C05358=1022.023,281.198,-131.885,170.057,49.076,159.456
C05359=1022.016,280.949,-131.855,170.053,49.079,159.456
C05360=1022.009,280.702,-131.824,170.047,49.082,159.456
C05361=1022.003,280.454,-131.794,170.043,49.086,159.456
C05362=1021.996,280.205,-131.763,170.039,49.089,159.456
C05363=1021.991,279.958,-131.733,170.034,49.092,159.456
C05364=1021.984,279.710,-131.701,170.030,49.095,159.456
C05365=1021.977,279.462,-131.671,170.024,49.099,159.456
C05366=1021.971,279.214,-131.641,170.020,49.102,159.456
C05367=1021.965,278.966,-131.610,170.015,49.105,159.456
C05368=1021.959,278.749,-131.583,170.011,49.108,159.456
C05369=1021.953,278.533,-131.557,170.008,49.111,159.456
C05370=1021.948,278.315,-131.529,170.003,49.114,159.456
C05371=1021.942,278.099,-131.503,169.999,49.117,159.456
C05372=1021.937,277.882,-131.477,169.995,49.120,159.456
C05373=1021.931,277.665,-131.450,169.991,49.122,159.456
C05374=1021.926,277.449,-131.423,169.987,49.126,159.457
C05375=1021.921,277.232,-131.396,169.983,49.129,159.457
C05376=1021.914,276.984,-131.366,169.979,49.132,159.457
C05377=1021.908,276.736,-131.336,169.974,49.136,159.457
C05378=1021.901,276.488,-131.306,169.969,49.138,159.457
C05379=1021.895,276.240,-131.275,169.964,49.142,159.457
C05380=1021.888,275.992,-131.244,169.960,49.146,159.457
C05381=1021.882,275.744,-131.215,169.955,49.149,159.457
C05382=1021.876,275.495,-131.185,169.951,49.153,159.457
C05383=1021.869,275.247,-131.155,169.946,49.156,159.457
C05384=1021.863,275.000,-131.125,169.942,49.160,159.457
C05385=1021.856,274.751,-131.094,169.938,49.163,159.457
C05386=1021.850,274.504,-131.064,169.933,49.167,159.457
C05387=1021.843,274.255,-131.034,169.929,49.170,159.457
C05388=1021.837,274.008,-131.004,169.923,49.173,159.457
C05389=1021.831,273.759,-130.974,169.919,49.177,159.458
C05390=1021.825,273.511,-130.944,169.914,49.181,159.458
C05391=1021.818,273.263,-130.914,169.910,49.184,159.458
C05392=1021.812,273.015,-130.883,169.905,49.187,159.458
C05393=1021.806,272.767,-130.853,169.901,49.191,159.458
C05394=1021.799,272.518,-130.824,169.896,49.195,159.458
C05395=1021.793,272.271,-130.794,169.892,49.198,159.458
C05396=1021.786,272.022,-130.763,169.887,49.202,159.458
C05397=1021.780,271.774,-130.734,169.883,49.206,159.458
C05398=1021.774,271.526,-130.704,169.879,49.209,159.459
C05399=1021.767,271.278,-130.674,169.874,49.213,159.459
C05400=1021.761,271.030,-130.644,169.870,49.216,159.459
C05401=1021.755,270.782,-130.614,169.865,49.220,159.459
C05402=1021.748,270.533,-130.584,169.861,49.223,159.459
C05403=1021.742,270.285,-130.555,169.856,49.227,159.459
C05404=1021.736,270.038,-130.525,169.852,49.231,159.459
C05405=1021.729,269.789,-130.495,169.847,49.235,159.459
C05406=1021.723,269.541,-130.465,169.843,49.238,159.460
C05407=1021.717,269.293,-130.435,169.838,49.242,159.460
C05408=1021.710,269.045,-130.405,169.834,49.246,159.460
C05409=1021.704,268.796,-130.376,169.829,49.250,159.460
C05410=1021.697,268.549,-130.346,169.825,49.253,159.460
C05411=1021.692,268.300,-130.317,169.821,49.257,159.460
C05412=1021.685,268.052,-130.287,169.816,49.260,159.460
C05413=1021.679,267.804,-130.258,169.812,49.264,159.460
C05414=1021.673,267.556,-130.227,169.807,49.268,159.461
C05415=1021.666,267.307,-130.198,169.803,49.271,159.461
C05416=1021.660,267.059,-130.169,169.799,49.276,159.461
C05417=1021.653,266.812,-130.139,169.795,49.279,159.461
C05418=1021.648,266.563,-130.109,169.790,49.283,159.461
C05419=1021.641,266.315,-130.080,169.786,49.287,159.461
C05420=1021.634,266.067,-130.050,169.781,49.291,159.462
C05421=1021.628,265.819,-130.021,169.777,49.294,159.462
C05422=1021.622,265.570,-129.992,169.772,49.298,159.462
C05423=1021.616,265.323,-129.962,169.768,49.302,159.462
C05424=1021.609,265.074,-129.932,169.763,49.306,159.462
C05425=1021.603,264.826,-129.903,169.759,49.310,159.462
C05426=1021.596,264.578,-129.874,169.754,49.314,159.463
C05427=1021.590,264.330,-129.845,169.751,49.318,159.463
C05428=1021.585,264.116,-129.819,169.747,49.321,159.463
C05429=1021.579,263.901,-129.794,169.742,49.324,159.463
C05430=1021.573,263.686,-129.769,169.739,49.328,159.463
C05431=1021.568,263.472,-129.744,169.735,49.331,159.463
C05432=1021.563,263.258,-129.718,169.731,49.335,159.464
C05433=1021.557,263.044,-129.693,169.728,49.338,159.464
C05434=1021.552,262.829,-129.668,169.724,49.341,159.464
C05435=1021.547,262.615,-129.643,169.720,49.345,159.464
C05436=1021.541,262.366,-129.614,169.716,49.349,159.464
C05437=1021.534,262.118,-129.584,169.712,49.352,159.464
C05438=1021.528,261.869,-129.555,169.708,49.357,159.465
C05439=1021.521,261.621,-129.526,169.703,49.360,159.465
C05440=1021.515,261.373,-129.497,169.699,49.365,159.465
C05441=1021.508,261.126,-129.467,169.694,49.369,159.465
C05442=1021.503,260.877,-129.438,169.690,49.372,159.466
C05443=1021.497,260.629,-129.409,169.686,49.377,159.466
C05444=1021.490,260.381,-129.380,169.682,49.380,159.466
C05445=1021.485,260.132,-129.351,169.677,49.385,159.466
C05446=1021.478,259.884,-129.323,169.673,49.388,159.466
C05447=1021.471,259.636,-129.294,169.669,49.393,159.467
C05448=1021.464,259.387,-129.265,169.665,49.397,159.467
C05449=1021.457,259.140,-129.236,169.660,49.401,159.467
C05450=1021.452,258.891,-129.208,169.656,49.405,159.468
C05451=1021.445,258.643,-129.179,169.652,49.410,159.468
C05452=1021.438,258.395,-129.150,169.647,49.414,159.468
C05453=1021.432,258.147,-129.121,169.643,49.418,159.468
C05454=1021.426,257.898,-129.093,169.639,49.422,159.469
C05455=1021.420,257.650,-129.064,169.635,49.426,159.469
C05456=1021.413,257.402,-129.035,169.630,49.430,159.469
C05457=1021.407,257.153,-129.007,169.626,49.435,159.469
C05458=1021.401,256.905,-128.978,169.622,49.439,159.470
C05459=1021.394,256.657,-128.950,169.618,49.443,159.470
C05460=1021.388,256.409,-128.921,169.613,49.447,159.470
C05461=1021.381,256.160,-128.892,169.610,49.452,159.470
C05462=1021.375,255.912,-128.865,169.605,49.456,159.471
C05463=1021.369,255.664,-128.835,169.601,49.460,159.471
C05464=1021.362,255.416,-128.806,169.596,49.464,159.471
C05465=1021.356,255.167,-128.779,169.592,49.469,159.471
C05466=1021.349,254.919,-128.750,169.588,49.473,159.472
C05467=1021.343,254.670,-128.721,169.583,49.477,159.472
C05468=1021.337,254.422,-128.692,169.580,49.481,159.472
C05469=1021.330,254.174,-128.665,169.575,49.486,159.473
C05470=1021.324,253.926,-128.636,169.571,49.490,159.473
C05471=1021.318,253.677,-128.607,169.567,49.494,159.473
C05472=1021.311,253.429,-128.579,169.563,49.499,159.474
C05473=1021.305,253.180,-128.550,169.559,49.503,159.474
C05474=1021.299,252.932,-128.521,169.555,49.507,159.474
C05475=1021.292,252.684,-128.494,169.550,49.511,159.474
C05476=1021.286,252.436,-128.465,169.546,49.516,159.475
C05477=1021.280,252.187,-128.436,169.542,49.520,159.475
C05478=1021.273,251.939,-128.408,169.538,49.524,159.475
C05479=1021.267,251.690,-128.380,169.534,49.529,159.476
C05480=1021.262,251.442,-128.352,169.530,49.533,159.476
C05481=1021.255,251.195,-128.323,169.525,49.538,159.476
C05482=1021.249,250.946,-128.295,169.522,49.542,159.477
C05483=1021.243,250.698,-128.266,169.517,49.547,159.477
C05484=1021.236,250.449,-128.238,169.513,49.551,159.477
C05485=1021.230,250.200,-128.210,169.509,49.555,159.477
C05486=1021.224,249.952,-128.181,169.504,49.560,159.478
C05487=1021.218,249.705,-128.153,169.501,49.564,159.478
C05488=1021.212,249.489,-128.128,169.497,49.568,159.478
C05489=1021.208,249.274,-128.104,169.493,49.572,159.479
C05490=1021.202,249.058,-128.080,169.490,49.575,159.479
C05491=1021.197,248.843,-128.055,169.487,49.579,159.479
C05492=1021.191,248.629,-128.030,169.483,49.583,159.479
C05493=1021.186,248.413,-128.006,169.479,49.587,159.480
C05494=1021.180,248.198,-127.982,169.475,49.591,159.480
C05495=1021.175,247.983,-127.957,169.473,49.595,159.480
C05496=1021.169,247.734,-127.929,169.468,49.599,159.481
C05497=1021.163,247.485,-127.901,169.464,49.604,159.481
C05498=1021.156,247.237,-127.872,169.460,49.608,159.481
C05499=1021.151,246.989,-127.844,169.456,49.612,159.482
C05500=1021.144,246.741,-127.816,169.452,49.617,159.482
C05501=1021.138,246.492,-127.788,169.448,49.621,159.482
C05502=1021.133,246.243,-127.760,169.443,49.626,159.483
C05503=1021.126,245.996,-127.732,169.440,49.630,159.483
C05504=1021.120,245.747,-127.703,169.435,49.635,159.483
C05505=1021.114,245.499,-127.675,169.432,49.640,159.484
C05506=1021.108,245.251,-127.648,169.427,49.644,159.484
C05507=1021.102,245.002,-127.619,169.424,49.648,159.484
C05508=1021.096,244.753,-127.591,169.419,49.653,159.485
C05509=1021.090,244.506,-127.564,169.415,49.657,159.485
C05510=1021.084,244.257,-127.535,169.411,49.662,159.485
C05511=1021.078,244.008,-127.507,169.408,49.667,159.486
C05512=1021.072,243.761,-127.479,169.403,49.671,159.486
C05513=1021.066,243.512,-127.451,169.399,49.676,159.486
C05514=1021.060,243.263,-127.423,169.395,49.681,159.487
C05515=1021.054,243.015,-127.395,169.392,49.685,159.487
C05516=1021.048,242.767,-127.368,169.387,49.690,159.487
C05517=1021.041,242.518,-127.340,169.383,49.695,159.488
C05518=1021.036,242.270,-127.312,169.379,49.699,159.488
C05519=1021.029,242.022,-127.284,169.375,49.704,159.489
C05520=1021.023,241.773,-127.256,169.371,49.709,159.489
C05521=1021.017,241.525,-127.229,169.367,49.713,159.489
C05522=1021.010,241.277,-127.201,169.364,49.718,159.490
C05523=1021.005,241.028,-127.173,169.359,49.723,159.490
C05524=1020.998,240.780,-127.146,169.355,49.728,159.491
C05525=1020.992,240.531,-127.118,169.351,49.732,159.491
C05526=1020.986,240.283,-127.090,169.347,49.737,159.491
C05527=1020.980,240.035,-127.063,169.343,49.742,159.492
C05528=1020.973,239.786,-127.036,169.339,49.746,159.492
C05529=1020.968,239.538,-127.008,169.336,49.751,159.493
C05530=1020.961,239.289,-126.980,169.331,49.756,159.493
C05531=1020.955,239.042,-126.952,169.327,49.761,159.493
C05532=1020.949,238.793,-126.925,169.324,49.766,159.494
C05533=1020.942,238.544,-126.898,169.319,49.771,159.494
C05534=1020.937,238.295,-126.870,169.316,49.776,159.495
C05535=1020.931,238.047,-126.843,169.311,49.780,159.495
C05536=1020.924,237.799,-126.815,169.307,49.785,159.496
C05537=1020.918,237.550,-126.788,169.304,49.790,159.496
C05538=1020.911,237.302,-126.761,169.299,49.795,159.496
C05539=1020.906,237.053,-126.734,169.296,49.800,159.497
C05540=1020.899,236.805,-126.706,169.292,49.805,159.497
C05541=1020.893,236.557,-126.680,169.287,49.810,159.498
C05542=1020.886,236.308,-126.652,169.284,49.815,159.498
C05543=1020.881,236.059,-126.625,169.280,49.820,159.499
C05544=1020.875,235.811,-126.597,169.275,49.825,159.499
C05545=1020.869,235.563,-126.570,169.272,49.830,159.499
C05546=1020.862,235.314,-126.543,169.268,49.835,159.500
C05547=1020.857,235.066,-126.516,169.264,49.840,159.500
C05548=1020.851,234.847,-126.492,169.261,49.844,159.501
C05549=1020.845,234.629,-126.468,169.257,49.848,159.501
C05550=1020.840,234.410,-126.444,169.254,49.853,159.502
C05551=1020.834,234.192,-126.421,169.251,49.858,159.502
C05552=1020.828,233.974,-126.396,169.247,49.862,159.502
C05553=1020.823,233.756,-126.373,169.243,49.866,159.503
C05554=1020.818,233.537,-126.348,169.240,49.871,159.503
C05555=1020.813,233.319,-126.325,169.237,49.875,159.504
C05556=1020.807,233.070,-126.298,169.232,49.881,159.504
C05557=1020.800,232.822,-126.270,169.229,49.885,159.504
C05558=1020.794,232.574,-126.244,169.225,49.890,159.505
C05559=1020.788,232.324,-126.217,169.220,49.895,159.505
C05560=1020.782,232.077,-126.189,169.217,49.900,159.506
C05561=1020.776,231.828,-126.162,169.213,49.906,159.506
C05562=1020.770,231.579,-126.136,169.209,49.911,159.507
C05563=1020.763,231.330,-126.109,169.206,49.916,159.507
C05564=1020.757,231.083,-126.081,169.201,49.921,159.508
C05565=1020.752,230.834,-126.055,169.198,49.926,159.508
C05566=1020.745,230.585,-126.027,169.194,49.931,159.509
C05567=1020.739,230.337,-126.000,169.189,49.936,159.509
C05568=1020.733,230.088,-125.973,169.186,49.941,159.510
C05569=1020.727,229.840,-125.946,169.182,49.946,159.510
C05570=1020.721,229.592,-125.920,169.178,49.952,159.511
C05571=1020.715,229.342,-125.893,169.175,49.957,159.511
C05572=1020.708,229.095,-125.866,169.171,49.962,159.512
C05573=1020.702,228.847,-125.839,169.167,49.968,159.512
C05574=1020.696,228.598,-125.812,169.163,49.973,159.513
C05575=1020.690,228.349,-125.786,169.159,49.978,159.513
C05576=1020.684,228.101,-125.759,169.155,49.983,159.514
C05577=1020.678,227.852,-125.732,169.152,49.988,159.514
C05578=1020.672,227.604,-125.705,169.148,49.994,159.515
C05579=1020.666,227.354,-125.678,169.143,49.999,159.515
C05580=1020.659,227.106,-125.652,169.140,50.004,159.516
C05581=1020.653,226.858,-125.626,169.136,50.009,159.516
C05582=1020.648,226.610,-125.599,169.132,50.015,159.517
C05583=1020.641,226.361,-125.572,169.129,50.020,159.517
C05584=1020.635,226.113,-125.546,169.125,50.025,159.518
C05585=1020.629,225.864,-125.519,169.120,50.031,159.518
C05586=1020.622,225.615,-125.493,169.117,50.037,159.519
C05587=1020.616,225.367,-125.466,169.113,50.042,159.520
C05588=1020.610,225.119,-125.440,169.109,50.047,159.520
C05589=1020.603,224.870,-125.413,169.105,50.053,159.521
C05590=1020.598,224.622,-125.387,169.101,50.058,159.521
C05591=1020.592,224.373,-125.361,169.098,50.063,159.522
C05592=1020.585,224.124,-125.334,169.094,50.068,159.522
C05593=1020.579,223.876,-125.308,169.090,50.074,159.523
C05594=1020.573,223.627,-125.281,169.086,50.080,159.523
C05595=1020.567,223.379,-125.255,169.083,50.085,159.524
C05596=1020.560,223.130,-125.228,169.079,50.091,159.524
C05597=1020.554,222.881,-125.202,169.075,50.096,159.525
C05598=1020.549,222.633,-125.176,169.071,50.102,159.526
C05599=1020.541,222.384,-125.149,169.068,50.107,159.526
C05600=1020.536,222.136,-125.123,169.063,50.112,159.527
C05601=1020.530,221.888,-125.096,169.060,50.118,159.527
C05602=1020.524,221.639,-125.071,169.057,50.123,159.528
C05603=1020.518,221.391,-125.044,169.053,50.129,159.528
C05604=1020.512,221.141,-125.017,169.049,50.135,159.529
C05605=1020.505,220.893,-124.991,169.045,50.141,159.530
C05606=1020.500,220.644,-124.965,169.042,50.146,159.530
C05607=1020.493,220.396,-124.939,169.037,50.151,159.531
C05608=1020.488,220.174,-124.915,169.034,50.156,159.531
C05609=1020.482,219.951,-124.891,169.031,50.161,159.532
C05610=1020.477,219.729,-124.868,169.027,50.166,159.532
C05611=1020.471,219.507,-124.845,169.024,50.171,159.533
C05612=1020.466,219.284,-124.822,169.020,50.176,159.533
C05613=1020.461,219.061,-124.798,169.017,50.181,159.534
C05614=1020.455,218.838,-124.774,169.014,50.186,159.534
C05615=1020.450,218.616,-124.751,169.011,50.191,159.535
C05616=1020.443,218.368,-124.725,169.007,50.196,159.535
C05617=1020.438,218.119,-124.699,169.003,50.202,159.536
C05618=1020.431,217.871,-124.673,168.999,50.208,159.537
C05619=1020.425,217.623,-124.647,168.996,50.213,159.537
C05620=1020.419,217.374,-124.621,168.992,50.219,159.538
C05621=1020.412,217.125,-124.595,168.988,50.225,159.538
C05622=1020.406,216.877,-124.569,168.984,50.231,159.539
C05623=1020.400,216.628,-124.543,168.980,50.237,159.540
C05624=1020.394,216.380,-124.517,168.977,50.243,159.540
C05625=1020.388,216.131,-124.492,168.974,50.248,159.541
C05626=1020.382,215.882,-124.466,168.970,50.254,159.541
C05627=1020.376,215.634,-124.440,168.966,50.260,159.542
C05628=1020.369,215.385,-124.414,168.962,50.266,159.543
C05629=1020.363,215.136,-124.387,168.958,50.272,159.543
C05630=1020.357,214.888,-124.362,168.954,50.277,159.544
C05631=1020.351,214.639,-124.337,168.951,50.283,159.545
C05632=1020.344,214.391,-124.311,168.947,50.289,159.545
C05633=1020.339,214.142,-124.285,168.944,50.295,159.546
C05634=1020.333,213.893,-124.259,168.940,50.301,159.547
C05635=1020.326,213.645,-124.233,168.936,50.306,159.547
C05636=1020.321,213.396,-124.207,168.932,50.312,159.548
C05637=1020.314,213.148,-124.182,168.929,50.318,159.548
C05638=1020.308,212.900,-124.156,168.925,50.324,159.549
C05639=1020.302,212.651,-124.130,168.922,50.330,159.550
C05640=1020.296,212.402,-124.105,168.918,50.336,159.550
C05641=1020.290,212.154,-124.079,168.914,50.341,159.551
C05642=1020.284,211.905,-124.053,168.910,50.347,159.551
C05643=1020.278,211.656,-124.027,168.907,50.353,159.552
C05644=1020.272,211.408,-124.002,168.903,50.359,159.553
C05645=1020.265,211.159,-123.976,168.900,50.365,159.553
C05646=1020.260,210.910,-123.950,168.896,50.371,159.554
C05647=1020.254,210.662,-123.925,168.892,50.377,159.555
C05648=1020.247,210.413,-123.899,168.888,50.383,159.555
C05649=1020.242,210.165,-123.873,168.885,50.389,159.556
C05650=1020.235,209.916,-123.847,168.882,50.395,159.557
C05651=1020.229,209.667,-123.822,168.878,50.401,159.557
C05652=1020.223,209.419,-123.797,168.874,50.407,159.558
C05653=1020.217,209.170,-123.771,168.870,50.413,159.559
C05654=1020.211,208.921,-123.746,168.867,50.419,159.559
C05655=1020.204,208.673,-123.721,168.863,50.425,159.560
C05656=1020.199,208.424,-123.695,168.859,50.431,159.561
C05657=1020.193,208.175,-123.669,168.855,50.437,159.561
C05658=1020.186,207.927,-123.643,168.852,50.443,159.562
C05659=1020.180,207.678,-123.618,168.849,50.449,159.563
C05660=1020.174,207.430,-123.593,168.845,50.455,159.564
C05661=1020.168,207.181,-123.567,168.841,50.461,159.564
C05662=1020.161,206.932,-123.542,168.838,50.468,159.565
C05663=1020.155,206.684,-123.517,168.834,50.474,159.566
C05664=1020.149,206.398,-123.488,168.830,50.481,159.566
C05665=1020.141,206.111,-123.459,168.825,50.488,159.567
C05666=1020.134,205.825,-123.429,168.821,50.495,159.568
C05667=1020.127,205.539,-123.401,168.818,50.502,159.569
C05668=1020.118,205.137,-123.360,168.811,50.512,159.570
C05669=1020.107,204.735,-123.320,168.805,50.522,159.571
C05670=1020.097,204.333,-123.279,168.800,50.532,159.572
C05671=1020.088,203.931,-123.238,168.794,50.542,159.573
C05672=1020.065,202.891,-123.139,168.342,50.448,159.476
C05673=1020.060,202.642,-123.116,168.337,50.455,159.477
C05674=1020.055,202.393,-123.093,168.333,50.463,159.478
C05675=1020.050,202.145,-123.068,168.329,50.470,159.479
C05676=1020.044,201.896,-123.045,168.324,50.477,159.479
C05677=1020.039,201.647,-123.022,168.320,50.484,159.480
C05678=1020.034,201.398,-122.998,168.316,50.492,159.481
C05679=1020.028,201.149,-122.975,168.311,50.499,159.482
C05680=1020.023,200.900,-122.951,168.307,50.506,159.482
C05681=1020.019,200.652,-122.928,168.302,50.513,159.483
C05682=1020.013,200.403,-122.904,168.298,50.520,159.484
C05683=1020.008,200.154,-122.881,168.294,50.528,159.485
C05684=1020.003,199.905,-122.857,168.289,50.535,159.485
C05685=1019.998,199.656,-122.834,168.285,50.542,159.486
C05686=1019.992,199.407,-122.811,168.280,50.549,159.487
C05687=1019.988,199.158,-122.788,168.276,50.557,159.488
C05688=1019.982,198.909,-122.765,168.272,50.564,159.488
C05689=1019.976,198.660,-122.742,168.267,50.571,159.489
C05690=1019.971,198.411,-122.718,168.263,50.579,159.490
C05691=1019.965,198.162,-122.695,168.259,50.586,159.491
C05692=1019.960,197.913,-122.672,168.255,50.593,159.491
C05693=1019.955,197.665,-122.649,168.251,50.601,159.492
C05694=1019.950,197.416,-122.626,168.246,50.608,159.493
C05695=1019.944,197.167,-122.603,168.242,50.615,159.494
C05696=1019.939,196.918,-122.580,168.238,50.623,159.495
C05697=1019.934,196.670,-122.557,168.233,50.630,159.495
C05698=1019.928,196.421,-122.534,168.229,50.637,159.496
C05699=1019.923,196.172,-122.511,168.225,50.645,159.497
C05700=1019.917,195.923,-122.488,168.220,50.652,159.498
C05701=1019.912,195.675,-122.465,168.216,50.659,159.498
C05702=1019.907,195.425,-122.442,168.212,50.667,159.499
C05703=1019.901,195.176,-122.419,168.207,50.674,159.500
C05704=1019.896,194.927,-122.396,168.203,50.681,159.501
C05705=1019.892,194.678,-122.373,168.199,50.689,159.502
C05706=1019.886,194.429,-122.350,168.195,50.696,159.502
C05707=1019.880,194.181,-122.327,168.190,50.704,159.503
C05708=1019.876,193.932,-122.304,168.186,50.711,159.504
C05709=1019.870,193.683,-122.281,168.182,50.718,159.505
C05710=1019.865,193.434,-122.259,168.178,50.726,159.505
C05711=1019.860,193.184,-122.235,168.173,50.733,159.506
C05712=1019.854,192.936,-122.213,168.169,50.740,159.507
C05713=1019.849,192.687,-122.190,168.165,50.748,159.508
C05714=1019.844,192.439,-122.167,168.160,50.755,159.508
C05715=1019.839,192.189,-122.145,168.156,50.763,159.509
C05716=1019.833,191.940,-122.122,168.152,50.770,159.510
C05717=1019.829,191.692,-122.098,168.148,50.777,159.511
C05718=1019.823,191.442,-122.076,168.144,50.785,159.512
C05719=1019.818,191.194,-122.053,168.139,50.792,159.512
C05720=1019.813,190.945,-122.030,168.135,50.800,159.513
C05721=1019.808,190.696,-122.007,168.132,50.806,159.514
C05722=1019.803,190.447,-121.985,168.127,50.814,159.515
C05723=1019.798,190.198,-121.962,168.123,50.821,159.516
C05724=1019.792,189.949,-121.939,168.119,50.828,159.516
C05725=1019.787,189.700,-121.917,168.115,50.836,159.517
C05726=1019.782,189.451,-121.893,168.110,50.843,159.518
C05727=1019.777,189.203,-121.871,168.106,50.851,159.519
C05728=1019.772,188.953,-121.849,168.102,50.858,159.520
C05729=1019.767,188.705,-121.825,168.098,50.866,159.520
C05730=1019.762,188.455,-121.803,168.094,50.872,159.521
C05731=1019.757,188.207,-121.781,168.090,50.880,159.522
C05732=1019.751,187.958,-121.758,168.086,50.887,159.523
C05733=1019.746,187.677,-121.732,168.081,50.896,159.524
C05734=1019.740,187.396,-121.706,168.077,50.904,159.525
C05735=1019.734,187.114,-121.681,168.072,50.912,159.525
C05736=1019.728,186.833,-121.656,168.068,50.921,159.526
C05737=1019.724,186.585,-121.632,168.063,50.928,159.527
C05738=1019.718,186.335,-121.610,168.059,50.935,159.528
C05739=1019.713,186.087,-121.588,168.056,50.943,159.529
C05740=1019.708,185.837,-121.565,168.052,50.950,159.529
C05741=1019.703,185.589,-121.542,168.047,50.957,159.530
C05742=1019.698,185.339,-121.520,168.043,50.965,159.531
C05743=1019.693,185.091,-121.497,168.039,50.972,159.532
C05744=1019.689,184.842,-121.475,168.036,50.980,159.533
C05745=1019.683,184.593,-121.452,168.031,50.987,159.533
C05746=1019.678,184.344,-121.430,168.027,50.994,159.534
C05747=1019.673,184.095,-121.407,168.023,51.002,159.535
C05748=1019.668,183.846,-121.385,168.020,51.009,159.536
C05749=1019.663,183.597,-121.362,168.016,51.017,159.537
C05750=1019.658,183.348,-121.339,168.011,51.024,159.537
C05751=1019.654,183.100,-121.317,168.007,51.031,159.538
C05752=1019.648,182.850,-121.295,168.004,51.039,159.539
C05753=1019.644,182.602,-121.272,168.000,51.046,159.540
C05754=1019.638,182.352,-121.250,167.996,51.054,159.541
C05755=1019.634,182.103,-121.228,167.991,51.061,159.541
C05756=1019.628,181.854,-121.206,167.988,51.068,159.542
C05757=1019.623,181.605,-121.183,167.984,51.076,159.543
C05758=1019.617,181.356,-121.161,167.980,51.083,159.544
C05759=1019.612,181.107,-121.140,167.976,51.091,159.545
C05760=1019.607,180.858,-121.117,167.972,51.098,159.546
C05761=1019.601,180.609,-121.096,167.968,51.106,159.547
C05762=1019.596,180.361,-121.074,167.964,51.114,159.547
C05763=1019.591,180.111,-121.052,167.960,51.122,159.548
C05764=1019.585,179.863,-121.031,167.957,51.129,159.549
C05765=1019.580,179.613,-121.009,167.953,51.137,159.550
C05766=1019.575,179.364,-120.987,167.949,51.145,159.551
C05767=1019.569,179.116,-120.965,167.944,51.152,159.552
C05768=1019.564,178.866,-120.943,167.940,51.160,159.553
C05769=1019.559,178.617,-120.921,167.936,51.168,159.553
C05770=1019.554,178.369,-120.900,167.932,51.176,159.554
C05771=1019.548,178.119,-120.878,167.929,51.182,159.555
C05772=1019.544,177.870,-120.857,167.925,51.190,159.556
C05773=1019.538,177.621,-120.835,167.921,51.198,159.557
C05774=1019.533,177.372,-120.813,167.917,51.205,159.558
C05775=1019.528,177.123,-120.791,167.913,51.213,159.559
C05776=1019.522,176.875,-120.770,167.909,51.221,159.559
C05777=1019.517,176.625,-120.748,167.906,51.229,159.561
C05778=1019.512,176.376,-120.726,167.902,51.236,159.561
C05779=1019.506,176.128,-120.705,167.898,51.244,159.562
C05780=1019.501,175.878,-120.682,167.894,51.252,159.563
C05781=1019.496,175.629,-120.662,167.889,51.259,159.564
C05782=1019.491,175.380,-120.640,167.887,51.267,159.565
C05783=1019.486,175.131,-120.618,167.883,51.275,159.566
C05784=1019.480,174.882,-120.597,167.879,51.282,159.566
C05785=1019.475,174.634,-120.575,167.874,51.290,159.567
C05786=1019.470,174.385,-120.553,167.871,51.297,159.568
C05787=1019.464,174.135,-120.532,167.868,51.305,159.569
C05788=1019.460,173.886,-120.510,167.863,51.312,159.570
C05789=1019.455,173.637,-120.488,167.859,51.320,159.571
C05790=1019.449,173.389,-120.467,167.856,51.328,159.572
C05791=1019.444,173.139,-120.445,167.852,51.336,159.573
C05792=1019.439,172.890,-120.423,167.848,51.343,159.573
C05793=1019.434,172.641,-120.402,167.844,51.351,159.574
C05794=1019.429,172.392,-120.380,167.841,51.359,159.575
C05795=1019.423,172.143,-120.359,167.837,51.366,159.576
C05796=1019.418,171.894,-120.338,167.833,51.374,159.577
C05797=1019.412,171.612,-120.313,167.830,51.382,159.578
C05798=1019.407,171.331,-120.289,167.825,51.391,159.579
C05799=1019.401,171.050,-120.265,167.820,51.400,159.580
C05800=1019.395,170.768,-120.241,167.817,51.408,159.581
C05801=1019.390,170.519,-120.219,167.813,51.416,159.582
C05802=1019.386,170.270,-120.198,167.808,51.423,159.582
C05803=1019.380,170.021,-120.176,167.805,51.431,159.583
C05804=1019.375,169.771,-120.154,167.802,51.439,159.584
C05805=1019.370,169.522,-120.133,167.797,51.446,159.585
C05806=1019.365,169.274,-120.112,167.794,51.454,159.586
C05807=1019.360,169.025,-120.090,167.790,51.462,159.587
C05808=1019.354,168.776,-120.069,167.787,51.470,159.588
C05809=1019.350,168.527,-120.047,167.783,51.477,159.589
C05810=1019.345,168.277,-120.026,167.779,51.484,159.589
C05811=1019.340,168.029,-120.005,167.775,51.492,159.590
C05812=1019.334,167.779,-119.983,167.772,51.499,159.591
C05813=1019.330,167.530,-119.962,167.768,51.507,159.592
C05814=1019.324,167.281,-119.940,167.764,51.515,159.593
C05815=1019.320,167.032,-119.919,167.761,51.522,159.594
C05816=1019.314,166.783,-119.898,167.757,51.530,159.595
C05817=1019.309,166.534,-119.877,167.754,51.538,159.596
C05818=1019.305,166.285,-119.855,167.750,51.545,159.596
C05819=1019.299,166.036,-119.834,167.746,51.553,159.597
C05820=1019.295,165.787,-119.812,167.743,51.561,159.598
C05821=1019.290,165.538,-119.791,167.739,51.568,159.599
C05822=1019.284,165.289,-119.770,167.736,51.575,159.600
C05823=1019.280,165.040,-119.749,167.732,51.583,159.601
C05824=1019.274,164.791,-119.728,167.728,51.591,159.602
C05825=1019.270,164.542,-119.706,167.725,51.598,159.603
C05826=1019.265,164.293,-119.685,167.721,51.606,159.603
C05827=1019.260,164.044,-119.664,167.718,51.614,159.604
C05828=1019.255,163.795,-119.642,167.714,51.621,159.605
C05829=1019.249,163.545,-119.621,167.711,51.629,159.606
C05830=1019.244,163.297,-119.599,167.707,51.637,159.607
C05831=1019.240,163.047,-119.578,167.703,51.644,159.608
C05832=1019.234,162.799,-119.557,167.700,51.652,159.609
C05833=1019.230,162.550,-119.536,167.696,51.660,159.610
C05834=1019.226,162.300,-119.515,167.693,51.667,159.610
C05835=1019.220,162.052,-119.494,167.689,51.675,159.611
C05836=1019.216,161.803,-119.473,167.686,51.682,159.612
C05837=1019.210,161.554,-119.451,167.682,51.690,159.613
C05838=1019.206,161.305,-119.430,167.679,51.697,159.614
C05839=1019.201,161.055,-119.409,167.675,51.704,159.615
C05840=1019.196,160.807,-119.388,167.672,51.712,159.616
C05841=1019.191,160.557,-119.367,167.668,51.720,159.617
C05842=1019.186,160.308,-119.346,167.665,51.727,159.617
C05843=1019.181,160.059,-119.324,167.661,51.735,159.618
C05844=1019.176,159.810,-119.303,167.658,51.743,159.619
C05845=1019.171,159.561,-119.283,167.654,51.750,159.620
C05846=1019.166,159.312,-119.261,167.651,51.758,159.621
C05847=1019.161,159.063,-119.240,167.647,51.766,159.622
C05848=1019.157,158.813,-119.219,167.644,51.773,159.623
C05849=1019.151,158.564,-119.198,167.640,51.781,159.624
C05850=1019.146,158.315,-119.178,167.637,51.789,159.625
C05851=1019.142,158.066,-119.157,167.634,51.796,159.626
C05852=1019.137,157.817,-119.137,167.630,51.804,159.626
C05853=1019.131,157.569,-119.115,167.627,51.812,159.627
C05854=1019.126,157.320,-119.095,167.623,51.820,159.628
C05855=1019.121,157.070,-119.074,167.619,51.827,159.629
C05856=1019.116,156.821,-119.054,167.616,51.835,159.630
C05857=1019.110,156.572,-119.033,167.612,51.843,159.631
C05858=1019.106,156.323,-119.012,167.610,51.851,159.632
C05859=1019.101,156.074,-118.991,167.606,51.859,159.633
C05860=1019.095,155.825,-118.971,167.602,51.867,159.634
C05861=1019.090,155.543,-118.948,167.598,51.875,159.635
C05862=1019.084,155.261,-118.924,167.595,51.884,159.636
C05863=1019.078,154.978,-118.901,167.590,51.892,159.637
C05864=1019.072,154.697,-118.878,167.587,51.901,159.638
C05865=1019.067,154.448,-118.858,167.583,51.909,159.639
C05866=1019.062,154.199,-118.837,167.580,51.917,159.640
C05867=1019.057,153.950,-118.816,167.576,51.925,159.641
C05868=1019.052,153.701,-118.795,167.574,51.933,159.642
C05869=1019.047,153.452,-118.775,167.570,51.941,159.643
C05870=1019.042,153.202,-118.755,167.566,51.949,159.644
C05871=1019.037,152.953,-118.735,167.563,51.956,159.644
C05872=1019.032,152.704,-118.714,167.559,51.964,159.645
C05873=1019.027,152.455,-118.694,167.556,51.971,159.646
C05874=1019.021,152.206,-118.673,167.552,51.979,159.647
C05875=1019.016,151.957,-118.653,167.549,51.987,159.648
C05876=1019.012,151.708,-118.633,167.546,51.995,159.649
C05877=1019.007,151.459,-118.613,167.543,52.003,159.650
C05878=1019.001,151.209,-118.592,167.539,52.011,159.651
C05879=1018.996,150.960,-118.571,167.535,52.019,159.652
C05880=1018.991,150.711,-118.551,167.532,52.027,159.653
C05881=1018.986,150.462,-118.531,167.529,52.035,159.654
C05882=1018.981,150.213,-118.511,167.525,52.042,159.655
C05883=1018.976,149.964,-118.490,167.522,52.050,159.655
C05884=1018.971,149.715,-118.470,167.519,52.057,159.656
C05885=1018.966,149.465,-118.450,167.515,52.065,159.657
C05886=1018.961,149.217,-118.430,167.512,52.073,159.658
C05887=1018.956,148.968,-118.409,167.509,52.081,159.659
C05888=1018.951,148.718,-118.389,167.506,52.089,159.660
C05889=1018.946,148.469,-118.369,167.502,52.097,159.661
C05890=1018.941,148.220,-118.349,167.499,52.105,159.662
C05891=1018.936,147.971,-118.328,167.495,52.113,159.663
C05892=1018.931,147.721,-118.308,167.493,52.120,159.664
C05893=1018.925,147.473,-118.288,167.488,52.128,159.665
C05894=1018.920,147.223,-118.269,167.486,52.135,159.666
C05895=1018.915,146.974,-118.248,167.482,52.144,159.667
C05896=1018.910,146.725,-118.228,167.479,52.151,159.668
C05897=1018.905,146.475,-118.208,167.475,52.159,159.669
C05898=1018.900,146.227,-118.188,167.473,52.167,159.670
C05899=1018.895,145.977,-118.168,167.469,52.175,159.671
C05900=1018.890,145.728,-118.147,167.466,52.183,159.672
C05901=1018.885,145.480,-118.127,167.462,52.191,159.672
C05902=1018.880,145.230,-118.108,167.460,52.199,159.673
C05903=1018.874,144.981,-118.087,167.456,52.207,159.674
C05904=1018.870,144.731,-118.067,167.453,52.214,159.675
C05905=1018.864,144.483,-118.048,167.449,52.222,159.676
C05906=1018.859,144.234,-118.028,167.446,52.231,159.677
C05907=1018.854,143.984,-118.008,167.443,52.238,159.678
C05908=1018.849,143.736,-117.989,167.439,52.246,159.679
C05909=1018.844,143.486,-117.969,167.436,52.254,159.680
C05910=1018.839,143.237,-117.948,167.433,52.262,159.681
C05911=1018.834,142.988,-117.929,167.430,52.270,159.682
C05912=1018.828,142.739,-117.909,167.426,52.278,159.683
C05913=1018.823,142.489,-117.889,167.423,52.286,159.684
C05914=1018.819,142.240,-117.869,167.420,52.294,159.685
C05915=1018.813,141.991,-117.850,167.417,52.302,159.686
C05916=1018.808,141.742,-117.830,167.413,52.310,159.687
C05917=1018.803,141.493,-117.809,167.410,52.317,159.688
C05918=1018.798,141.244,-117.790,167.407,52.325,159.689
C05919=1018.793,140.994,-117.770,167.404,52.333,159.690
C05920=1018.788,140.746,-117.750,167.401,52.341,159.691
C05921=1018.782,140.496,-117.731,167.397,52.349,159.692
C05922=1018.777,140.247,-117.711,167.395,52.357,159.693
C05923=1018.773,139.998,-117.691,167.391,52.365,159.694
C05924=1018.768,139.748,-117.671,167.388,52.373,159.695
C05925=1018.761,139.386,-117.643,167.383,52.384,159.696
C05926=1018.753,139.023,-117.614,167.379,52.396,159.697
C05927=1018.745,138.661,-117.585,167.373,52.407,159.698
C05928=1018.738,138.298,-117.557,167.369,52.418,159.700
C05929=1018.733,138.048,-117.537,167.366,52.426,159.701
C05930=1018.728,137.799,-117.517,167.363,52.434,159.702
C05931=1018.723,137.550,-117.498,167.360,52.442,159.703
C05932=1018.718,137.301,-117.478,167.356,52.450,159.704
C05933=1018.713,137.052,-117.459,167.353,52.458,159.705
C05934=1018.708,136.802,-117.439,167.350,52.466,159.706
C05935=1018.703,136.554,-117.420,167.347,52.474,159.707
C05936=1018.698,136.304,-117.400,167.343,52.482,159.708
C05937=1018.692,136.054,-117.381,167.341,52.490,159.709
C05938=1018.688,135.805,-117.361,167.337,52.498,159.710
C05939=1018.682,135.556,-117.341,167.334,52.506,159.711
C05940=1018.677,135.307,-117.322,167.332,52.513,159.712
C05941=1018.672,135.058,-117.303,167.328,52.522,159.713
C05942=1018.667,134.809,-117.283,167.325,52.529,159.714
C05943=1018.662,134.560,-117.264,167.321,52.537,159.714
C05944=1018.657,134.311,-117.245,167.319,52.546,159.716
C05945=1018.648,133.893,-117.212,167.313,52.559,159.717
C05946=1018.639,133.475,-117.180,167.308,52.572,159.719
C05947=1018.631,133.057,-117.148,167.303,52.586,159.720
C05948=1018.623,132.640,-117.115,167.297,52.599,159.722
C05949=1018.617,132.391,-117.096,167.294,52.607,159.723
C05950=1018.613,132.142,-117.076,167.292,52.615,159.724
C05951=1018.607,131.892,-117.057,167.288,52.623,159.725
C05952=1018.602,131.643,-117.038,167.286,52.631,159.726
C05953=1018.597,131.394,-117.018,167.282,52.639,159.727
C05954=1018.592,131.145,-117.000,167.279,52.647,159.728
C05955=1018.587,130.895,-116.980,167.276,52.655,159.729
C05956=1018.582,130.646,-116.961,167.273,52.663,159.730
C05957=1018.576,130.397,-116.942,167.270,52.671,159.731
C05958=1018.572,130.148,-116.922,167.267,52.679,159.732
C05959=1018.566,129.899,-116.903,167.264,52.687,159.733
C05960=1018.562,129.650,-116.883,167.260,52.695,159.734
C05961=1018.556,129.400,-116.864,167.258,52.703,159.735
C05962=1018.552,129.151,-116.846,167.254,52.711,159.736
C05963=1018.546,128.901,-116.827,167.251,52.719,159.737
C05964=1018.541,128.653,-116.808,167.248,52.727,159.738
C05965=1018.536,128.404,-116.789,167.245,52.735,159.739
C05966=1018.530,128.154,-116.771,167.242,52.744,159.740
C05967=1018.525,127.905,-116.752,167.239,52.751,159.741
C05968=1018.520,127.656,-116.732,167.235,52.760,159.742
C05969=1018.514,127.407,-116.714,167.233,52.767,159.743
C05970=1018.509,127.157,-116.695,167.229,52.776,159.744
C05971=1018.504,126.908,-116.676,167.227,52.784,159.745
C05972=1018.499,126.658,-116.656,167.223,52.792,159.746
C05973=1018.494,126.409,-116.638,167.221,52.800,159.747
C05974=1018.489,126.160,-116.619,167.217,52.808,159.748
C05975=1018.483,125.911,-116.600,167.214,52.816,159.749
C05976=1018.479,125.661,-116.582,167.212,52.824,159.750
C05977=1018.473,125.412,-116.563,167.209,52.833,159.751
C05978=1018.468,125.163,-116.544,167.206,52.841,159.752
C05979=1018.463,124.914,-116.526,167.202,52.849,159.753
C05980=1018.457,124.665,-116.506,167.200,52.857,159.754
C05981=1018.452,124.416,-116.487,167.196,52.865,159.755
C05982=1018.447,124.166,-116.469,167.193,52.873,159.756
C05983=1018.442,123.917,-116.450,167.190,52.881,159.757
C05984=1018.437,123.668,-116.431,167.187,52.889,159.758
C05985=1018.431,123.386,-116.410,167.184,52.898,159.759
C05986=1018.425,123.104,-116.389,167.180,52.908,159.760
C05987=1018.419,122.822,-116.368,167.177,52.916,159.761
C05988=1018.414,122.540,-116.346,167.174,52.925,159.762
C05989=1018.409,122.290,-116.327,167.170,52.934,159.763
C05990=1018.403,122.041,-116.309,167.167,52.941,159.764
C05991=1018.399,121.792,-116.290,167.165,52.950,159.766
C05992=1018.393,121.542,-116.271,167.162,52.958,159.766
C05993=1018.388,121.293,-116.253,167.159,52.966,159.767
C05994=1018.383,121.044,-116.234,167.155,52.974,159.768
C05995=1018.377,120.795,-116.215,167.153,52.982,159.769
C05996=1018.373,120.546,-116.197,167.150,52.990,159.770
C05997=1018.368,120.297,-116.178,167.147,52.998,159.771
C05998=1018.362,120.047,-116.159,167.144,53.006,159.772
C05999=1018.357,119.798,-116.140,167.140,53.014,159.773
C06000=1018.353,119.548,-116.122,167.138,53.022,159.774
C06001=1018.347,119.299,-116.102,167.135,53.030,159.775
C06002=1018.343,119.050,-116.084,167.132,53.038,159.776
C06003=1018.338,118.801,-116.065,167.129,53.046,159.777
C06004=1018.333,118.552,-116.047,167.126,53.054,159.778
C06005=1018.327,118.302,-116.028,167.123,53.063,159.779
C06006=1018.322,118.053,-116.010,167.121,53.070,159.780
C06007=1018.317,117.804,-115.991,167.117,53.079,159.781
C06008=1018.312,117.555,-115.973,167.114,53.087,159.782
C06009=1018.307,117.305,-115.954,167.112,53.094,159.783
C06010=1018.302,117.056,-115.935,167.108,53.103,159.784
C06011=1018.297,116.807,-115.916,167.106,53.111,159.785
C06012=1018.292,116.558,-115.898,167.103,53.118,159.786
C06013=1018.287,116.308,-115.880,167.099,53.127,159.787
C06014=1018.282,116.059,-115.861,167.097,53.134,159.788
C06015=1018.277,115.810,-115.843,167.094,53.142,159.789
C06016=1018.272,115.561,-115.824,167.091,53.151,159.790
C06017=1018.266,115.311,-115.805,167.088,53.158,159.791
C06018=1018.261,115.062,-115.786,167.086,53.166,159.792
C06019=1018.256,114.813,-115.768,167.082,53.175,159.793
C06020=1018.252,114.563,-115.750,167.079,53.182,159.794
C06021=1018.247,114.315,-115.731,167.077,53.190,159.795
C06022=1018.242,114.064,-115.712,167.074,53.198,159.796
C06023=1018.237,113.815,-115.694,167.071,53.206,159.797
C06024=1018.232,113.566,-115.675,167.068,53.214,159.798
C06025=1018.227,113.317,-115.657,167.066,53.222,159.799
C06026=1018.222,113.068,-115.638,167.062,53.230,159.800
C06027=1018.217,112.819,-115.620,167.059,53.238,159.801
C06028=1018.212,112.569,-115.601,167.056,53.245,159.802
C06029=1018.207,112.320,-115.583,167.054,53.253,159.803
C06030=1018.202,112.071,-115.564,167.050,53.262,159.804
C06031=1018.197,111.822,-115.547,167.048,53.270,159.805
C06032=1018.192,111.572,-115.529,167.045,53.278,159.806
C06033=1018.187,111.322,-115.510,167.042,53.286,159.807
C06034=1018.181,111.074,-115.491,167.040,53.294,159.808
C06035=1018.176,110.824,-115.474,167.036,53.302,159.809
C06036=1018.171,110.575,-115.455,167.033,53.310,159.810
C06037=1018.166,110.326,-115.437,167.031,53.318,159.811
C06038=1018.162,110.076,-115.419,167.027,53.327,159.812
C06039=1018.155,109.827,-115.401,167.025,53.334,159.813
C06040=1018.151,109.577,-115.383,167.022,53.343,159.814
C06041=1018.146,109.329,-115.364,167.019,53.351,159.815
C06042=1018.140,109.080,-115.347,167.017,53.359,159.816
C06043=1018.135,108.830,-115.328,167.013,53.367,159.817
C06044=1018.131,108.581,-115.310,167.010,53.375,159.818
C06045=1018.125,108.332,-115.293,167.007,53.384,159.819
C06046=1018.120,108.082,-115.274,167.005,53.392,159.820
C06047=1018.114,107.833,-115.257,167.002,53.400,159.821
C06048=1018.109,107.583,-115.238,166.999,53.408,159.822
C06049=1018.104,107.301,-115.218,166.996,53.417,159.823
C06050=1018.098,107.019,-115.199,166.993,53.426,159.825
C06051=1018.092,106.737,-115.178,166.990,53.436,159.826
C06052=1018.086,106.455,-115.158,166.986,53.445,159.827
C06053=1018.081,106.206,-115.139,166.983,53.453,159.828
C06054=1018.075,105.956,-115.122,166.981,53.461,159.829
C06055=1018.071,105.707,-115.104,166.977,53.470,159.830
C06056=1018.065,105.458,-115.086,166.975,53.477,159.831
C06057=1018.060,105.209,-115.068,166.972,53.486,159.832
C06058=1018.055,104.960,-115.050,166.969,53.494,159.833
C06059=1018.050,104.710,-115.032,166.967,53.502,159.834
C06060=1018.045,104.461,-115.014,166.963,53.511,159.835
C06061=1018.040,104.212,-114.997,166.961,53.519,159.836
C06062=1018.035,103.961,-114.979,166.958,53.526,159.837
C06063=1018.029,103.712,-114.961,166.955,53.535,159.838
C06064=1018.024,103.463,-114.943,166.952,53.543,159.839
C06065=1018.019,103.214,-114.925,166.950,53.551,159.840
C06066=1018.014,102.965,-114.907,166.946,53.559,159.841
C06067=1018.009,102.715,-114.890,166.944,53.568,159.842
C06068=1018.004,102.466,-114.872,166.942,53.575,159.843
C06069=1017.998,102.217,-114.854,166.938,53.584,159.844
C06070=1017.993,101.968,-114.836,166.936,53.592,159.845
C06071=1017.989,101.718,-114.818,166.933,53.600,159.846
C06072=1017.983,101.469,-114.801,166.930,53.608,159.847
C06073=1017.979,101.219,-114.783,166.927,53.616,159.848
C06074=1017.973,100.970,-114.765,166.925,53.624,159.849
C06075=1017.968,100.721,-114.747,166.921,53.632,159.850
C06076=1017.963,100.472,-114.729,166.919,53.640,159.851
C06077=1017.958,100.223,-114.711,166.916,53.648,159.852
C06078=1017.953,99.973,-114.694,166.913,53.656,159.853
C06079=1017.948,99.724,-114.676,166.910,53.664,159.854
C06080=1017.943,99.475,-114.659,166.908,53.672,159.855
C06081=1017.938,99.225,-114.640,166.905,53.680,159.856
C06082=1017.933,98.976,-114.624,166.902,53.688,159.857
C06083=1017.928,98.726,-114.605,166.900,53.697,159.859
C06084=1017.922,98.477,-114.588,166.896,53.705,159.860
C06085=1017.917,98.227,-114.571,166.894,53.713,159.861
C06086=1017.912,97.978,-114.553,166.891,53.721,159.862
C06087=1017.907,97.729,-114.535,166.888,53.730,159.863
C06088=1017.902,97.479,-114.518,166.886,53.738,159.864
C06089=1017.896,97.230,-114.501,166.882,53.747,159.865
C06090=1017.891,96.981,-114.483,166.880,53.755,159.866
C06091=1017.886,96.731,-114.466,166.877,53.763,159.867
C06092=1017.881,96.482,-114.448,166.874,53.771,159.868
C06093=1017.875,96.233,-114.431,166.871,53.779,159.869
C06094=1017.870,95.984,-114.414,166.869,53.788,159.870
C06095=1017.865,95.734,-114.396,166.866,53.796,159.871
C06096=1017.860,95.485,-114.379,166.864,53.804,159.872
C06097=1017.854,95.236,-114.361,166.860,53.812,159.873
C06098=1017.849,94.986,-114.344,166.858,53.820,159.874
C06099=1017.845,94.737,-114.327,166.855,53.828,159.875
C06100=1017.840,94.488,-114.310,166.852,53.837,159.876
C06101=1017.834,94.239,-114.292,166.849,53.844,159.877
C06102=1017.829,93.989,-114.275,166.847,53.853,159.878
C06103=1017.824,93.740,-114.257,166.844,53.862,159.879
C06104=1017.819,93.491,-114.240,166.841,53.869,159.880
C06105=1017.813,93.241,-114.223,166.839,53.877,159.881
C06106=1017.808,92.992,-114.205,166.836,53.886,159.882
C06107=1017.803,92.742,-114.188,166.833,53.894,159.883
C06108=1017.798,92.493,-114.170,166.831,53.902,159.884
C06109=1017.793,92.243,-114.153,166.827,53.910,159.885
C06110=1017.788,91.995,-114.136,166.825,53.918,159.886
C06111=1017.783,91.745,-114.119,166.822,53.926,159.887
C06112=1017.778,91.496,-114.101,166.819,53.934,159.888
C06113=1017.772,91.214,-114.083,166.816,53.944,159.890
C06114=1017.766,90.931,-114.062,166.813,53.953,159.891
C06115=1017.760,90.650,-114.043,166.810,53.962,159.892
C06116=1017.755,90.368,-114.024,166.807,53.971,159.893
C06117=1017.750,90.119,-114.005,166.805,53.979,159.894
C06118=1017.745,89.869,-113.989,166.802,53.988,159.895
C06119=1017.739,89.619,-113.972,166.799,53.996,159.896
C06120=1017.734,89.370,-113.954,166.797,54.004,159.897
C06121=1017.729,89.120,-113.937,166.793,54.012,159.898
C06122=1017.724,88.872,-113.920,166.791,54.020,159.899
C06123=1017.719,88.622,-113.903,166.789,54.028,159.900
C06124=1017.714,88.373,-113.886,166.785,54.037,159.901
C06125=1017.709,88.123,-113.869,166.783,54.045,159.902
C06126=1017.703,87.874,-113.852,166.781,54.053,159.903
C06127=1017.697,87.625,-113.835,166.777,54.062,159.904
C06128=1017.692,87.375,-113.818,166.775,54.070,159.905
C06129=1017.688,87.126,-113.802,166.772,54.078,159.906
C06130=1017.682,86.877,-113.784,166.770,54.087,159.908
C06131=1017.677,86.627,-113.767,166.767,54.095,159.909
C06132=1017.672,86.378,-113.751,166.764,54.103,159.910
C06133=1017.666,86.128,-113.734,166.761,54.111,159.911
C06134=1017.661,85.880,-113.717,166.758,54.120,159.912
C06135=1017.656,85.630,-113.700,166.756,54.128,159.913
C06136=1017.651,85.380,-113.683,166.753,54.136,159.914
C06137=1017.646,85.131,-113.666,166.750,54.145,159.915
C06138=1017.641,84.881,-113.649,166.748,54.153,159.916
C06139=1017.636,84.632,-113.633,166.746,54.161,159.917
C06140=1017.630,84.383,-113.616,166.742,54.169,159.918
C06141=1017.625,84.134,-113.599,166.740,54.177,159.919
C06142=1017.619,83.884,-113.582,166.737,54.185,159.920
C06143=1017.614,83.634,-113.565,166.734,54.194,159.921
C06144=1017.609,83.385,-113.549,166.732,54.202,159.922
C06145=1017.604,83.136,-113.532,166.729,54.211,159.923
C06146=1017.599,82.887,-113.514,166.726,54.219,159.924
C06147=1017.594,82.637,-113.497,166.724,54.227,159.925
C06148=1017.589,82.388,-113.481,166.721,54.235,159.926
C06149=1017.584,82.139,-113.464,166.718,54.243,159.927
C06150=1017.579,81.889,-113.447,166.716,54.251,159.928
C06151=1017.573,81.639,-113.430,166.712,54.260,159.929
C06152=1017.568,81.391,-113.414,166.710,54.268,159.930
C06153=1017.563,81.141,-113.398,166.708,54.276,159.931
C06154=1017.557,80.892,-113.380,166.705,54.284,159.932
C06155=1017.552,80.642,-113.363,166.702,54.292,159.933
C06156=1017.547,80.393,-113.347,166.700,54.300,159.934
C06157=1017.542,80.144,-113.330,166.697,54.308,159.935
C06158=1017.537,79.894,-113.313,166.694,54.317,159.936
C06159=1017.532,79.645,-113.296,166.692,54.325,159.937
C06160=1017.527,79.395,-113.280,166.689,54.333,159.938
C06161=1017.522,79.146,-113.263,166.686,54.341,159.939
C06162=1017.517,78.896,-113.246,166.683,54.349,159.940
C06163=1017.511,78.647,-113.230,166.681,54.357,159.941
C06164=1017.506,78.398,-113.213,166.679,54.365,159.943
C06165=1017.501,78.148,-113.196,166.675,54.374,159.943
C06166=1017.496,77.899,-113.180,166.673,54.382,159.944
C06167=1017.491,77.649,-113.163,166.671,54.390,159.946
C06168=1017.486,77.400,-113.146,166.667,54.398,159.946
C06169=1017.481,77.151,-113.130,166.665,54.406,159.948
C06170=1017.476,76.901,-113.113,166.663,54.414,159.949
C06171=1017.470,76.652,-113.097,166.660,54.423,159.950
C06172=1017.466,76.403,-113.080,166.658,54.431,159.951
C06173=1017.460,76.153,-113.063,166.655,54.440,159.952
C06174=1017.455,75.903,-113.046,166.652,54.448,159.953
C06175=1017.450,75.655,-113.030,166.650,54.456,159.954
C06176=1017.445,75.405,-113.014,166.647,54.464,159.955
C06177=1017.439,75.123,-112.995,166.643,54.474,159.956
C06178=1017.433,74.841,-112.977,166.640,54.483,159.957
C06179=1017.427,74.559,-112.958,166.638,54.492,159.958
C06180=1017.421,74.277,-112.940,166.635,54.502,159.960
C06181=1017.416,74.028,-112.924,166.633,54.510,159.961
C06182=1017.411,73.779,-112.907,166.630,54.518,159.962
C06183=1017.405,73.529,-112.891,166.627,54.526,159.963
C06184=1017.400,73.280,-112.874,166.624,54.535,159.964
C06185=1017.395,73.030,-112.859,166.622,54.543,159.965
C06186=1017.390,72.781,-112.842,166.619,54.551,159.966
C06187=1017.385,72.532,-112.825,166.616,54.559,159.967
C06188=1017.379,72.282,-112.809,166.614,54.568,159.968
C06189=1017.374,72.033,-112.793,166.611,54.576,159.969
C06190=1017.369,71.783,-112.777,166.608,54.584,159.970
C06191=1017.364,71.535,-112.761,166.606,54.592,159.971
C06192=1017.359,71.285,-112.744,166.603,54.600,159.972
C06193=1017.353,71.035,-112.728,166.600,54.609,159.973
C06194=1017.348,70.786,-112.712,166.598,54.617,159.974
C06195=1017.343,70.536,-112.695,166.596,54.625,159.975
C06196=1017.338,70.288,-112.679,166.592,54.633,159.976
C06197=1017.333,70.037,-112.663,166.590,54.641,159.977
C06198=1017.327,69.788,-112.647,166.588,54.649,159.978
C06199=1017.322,69.539,-112.630,166.585,54.658,159.979
C06200=1017.317,69.289,-112.615,166.582,54.666,159.980
C06201=1017.312,69.040,-112.598,166.580,54.674,159.981
C06202=1017.307,68.790,-112.581,166.577,54.682,159.982
C06203=1017.302,68.541,-112.566,166.574,54.691,159.983
C06204=1017.297,68.292,-112.549,166.572,54.699,159.984
C06205=1017.291,68.043,-112.533,166.570,54.707,159.985
C06206=1017.286,67.793,-112.517,166.567,54.716,159.986
C06207=1017.280,67.543,-112.501,166.565,54.724,159.988
C06208=1017.276,67.294,-112.485,166.562,54.732,159.989
C06209=1017.270,67.044,-112.469,166.559,54.741,159.989
C06210=1017.265,66.795,-112.454,166.557,54.749,159.991
C06211=1017.260,66.545,-112.437,166.553,54.757,159.991
C06212=1017.255,66.296,-112.422,166.551,54.765,159.993
C06213=1017.250,66.046,-112.405,166.549,54.774,159.994
C06214=1017.244,65.798,-112.389,166.546,54.782,159.995
C06215=1017.239,65.548,-112.373,166.543,54.790,159.996
C06216=1017.234,65.299,-112.357,166.541,54.798,159.997
C06217=1017.228,65.049,-112.341,166.538,54.807,159.998
C06218=1017.224,64.800,-112.325,166.536,54.815,159.999
C06219=1017.218,64.550,-112.309,166.533,54.823,160.000
C06220=1017.213,64.301,-112.294,166.530,54.831,160.001
C06221=1017.208,64.051,-112.277,166.528,54.840,160.002
C06222=1017.203,63.802,-112.262,166.526,54.848,160.003
C06223=1017.198,63.552,-112.245,166.522,54.856,160.004
C06224=1017.193,63.303,-112.230,166.520,54.864,160.005
C06225=1017.187,63.054,-112.214,166.518,54.872,160.006
C06226=1017.182,62.804,-112.198,166.515,54.881,160.007
C06227=1017.177,62.554,-112.183,166.512,54.889,160.008
C06228=1017.171,62.305,-112.167,166.510,54.898,160.009
C06229=1017.166,62.055,-112.151,166.507,54.906,160.010
C06230=1017.161,61.806,-112.136,166.504,54.915,160.011
C06231=1017.155,61.556,-112.120,166.502,54.923,160.012
C06232=1017.150,61.307,-112.105,166.500,54.931,160.013
C06233=1017.144,61.058,-112.089,166.496,54.940,160.014
C06234=1017.139,60.808,-112.074,166.495,54.948,160.016
C06235=1017.133,60.558,-112.058,166.491,54.957,160.016
C06236=1017.129,60.309,-112.042,166.489,54.965,160.018
C06237=1017.124,60.060,-112.027,166.486,54.974,160.018
C06238=1017.118,59.810,-112.011,166.484,54.982,160.020
C06239=1017.113,59.561,-111.996,166.480,54.990,160.020
C06240=1017.107,59.311,-111.980,166.478,54.998,160.022
C06241=1017.102,59.030,-111.963,166.476,55.008,160.023
C06242=1017.095,58.748,-111.945,166.473,55.018,160.024
C06243=1017.089,58.465,-111.927,166.469,55.027,160.025
C06244=1017.083,58.184,-111.910,166.467,55.037,160.026
C06245=1017.078,57.934,-111.894,166.464,55.045,160.027
C06246=1017.073,57.685,-111.879,166.461,55.053,160.028
C06247=1017.067,57.435,-111.864,166.459,55.061,160.029
C06248=1017.062,57.186,-111.848,166.456,55.070,160.030
C06249=1017.057,56.937,-111.833,166.454,55.078,160.032
C06250=1017.051,56.687,-111.817,166.451,55.086,160.033
C06251=1017.046,56.438,-111.802,166.448,55.095,160.034
C06252=1017.041,56.189,-111.787,166.446,55.104,160.035
C06253=1017.035,55.939,-111.771,166.443,55.112,160.036
C06254=1017.030,55.689,-111.756,166.441,55.120,160.037
C06255=1017.025,55.440,-111.740,166.439,55.128,160.038
C06256=1017.019,55.191,-111.724,166.436,55.137,160.039
C06257=1017.014,54.942,-111.709,166.433,55.145,160.040
C06258=1017.009,54.692,-111.694,166.430,55.154,160.041
C06259=1017.004,54.442,-111.679,166.428,55.162,160.042
C06260=1016.999,54.193,-111.663,166.426,55.170,160.043
C06261=1016.994,53.943,-111.647,166.423,55.179,160.044
C06262=1016.989,53.694,-111.632,166.420,55.187,160.045
C06263=1016.984,53.444,-111.617,166.418,55.195,160.046
C06264=1016.978,53.194,-111.601,166.415,55.203,160.047
C06265=1016.973,52.945,-111.586,166.412,55.211,160.048
C06266=1016.968,52.696,-111.571,166.410,55.219,160.049
C06267=1016.962,52.446,-111.555,166.407,55.228,160.050
C06268=1016.957,52.197,-111.540,166.405,55.236,160.051
C06269=1016.952,51.948,-111.524,166.403,55.244,160.052
C06270=1016.946,51.698,-111.509,166.399,55.253,160.053
C06271=1016.941,51.449,-111.494,166.397,55.261,160.054
C06272=1016.936,51.199,-111.479,166.394,55.269,160.055
C06273=1016.930,50.949,-111.463,166.392,55.277,160.056
C06274=1016.925,50.700,-111.448,166.390,55.286,160.057
C06275=1016.920,50.451,-111.433,166.388,55.294,160.058
C06276=1016.915,50.202,-111.417,166.384,55.302,160.059
C06277=1016.910,49.952,-111.402,166.382,55.310,160.060
C06278=1016.905,49.702,-111.387,166.380,55.318,160.061
C06279=1016.900,49.453,-111.372,166.376,55.327,160.062
C06280=1016.894,49.203,-111.356,166.374,55.335,160.063
C06281=1016.889,48.954,-111.341,166.372,55.343,160.064
C06282=1016.885,48.704,-111.325,166.369,55.351,160.065
C06283=1016.880,48.455,-111.310,166.367,55.360,160.066
C06284=1016.874,48.205,-111.294,166.364,55.367,160.067
C06285=1016.869,47.956,-111.279,166.361,55.376,160.068
C06286=1016.864,47.707,-111.264,166.359,55.384,160.069
C06287=1016.859,47.457,-111.250,166.357,55.392,160.070
C06288=1016.853,47.207,-111.234,166.353,55.401,160.071
C06289=1016.848,46.957,-111.219,166.351,55.408,160.072
C06290=1016.843,46.708,-111.204,166.349,55.416,160.073
C06291=1016.838,46.459,-111.189,166.347,55.424,160.074
C06292=1016.833,46.210,-111.173,166.343,55.433,160.075
C06293=1016.828,45.960,-111.158,166.341,55.441,160.076
C06294=1016.823,45.710,-111.143,166.339,55.449,160.077
C06295=1016.817,45.461,-111.127,166.337,55.457,160.078
C06296=1016.812,45.212,-111.112,166.333,55.466,160.079
C06297=1016.807,44.963,-111.097,166.331,55.474,160.080
C06298=1016.802,44.713,-111.082,166.329,55.481,160.081
C06299=1016.797,44.463,-111.067,166.325,55.490,160.082
C06300=1016.792,44.213,-111.052,166.323,55.498,160.083
C06301=1016.787,43.964,-111.037,166.321,55.506,160.084
C06302=1016.782,43.715,-111.022,166.319,55.514,160.085
C06303=1016.776,43.465,-111.006,166.315,55.522,160.086
C06304=1016.771,43.216,-110.991,166.313,55.531,160.087
C06305=1016.766,42.934,-110.974,166.310,55.539,160.088
C06306=1016.760,42.652,-110.957,166.308,55.548,160.089
C06307=1016.754,42.370,-110.940,166.305,55.558,160.090
C06308=1016.749,42.088,-110.923,166.302,55.566,160.091
C06309=1016.744,41.839,-110.908,166.300,55.575,160.093
C06310=1016.738,41.588,-110.893,166.297,55.583,160.093
C06311=1016.733,41.339,-110.878,166.294,55.591,160.095
C06312=1016.728,41.090,-110.863,166.292,55.600,160.096
C06313=1016.723,40.840,-110.849,166.289,55.608,160.097
C06314=1016.717,40.591,-110.834,166.287,55.616,160.097
C06315=1016.712,40.342,-110.819,166.285,55.624,160.099
C06316=1016.707,40.092,-110.804,166.281,55.633,160.099
C06317=1016.702,39.842,-110.789,166.279,55.641,160.101
C06318=1016.696,39.593,-110.774,166.277,55.649,160.102
C06319=1016.691,39.343,-110.760,166.274,55.658,160.103
C06320=1016.686,39.094,-110.745,166.271,55.665,160.103
C06321=1016.681,38.844,-110.731,166.269,55.673,160.105
C06322=1016.676,38.595,-110.716,166.266,55.682,160.106
C06323=1016.671,38.346,-110.700,166.264,55.690,160.107
C06324=1016.666,38.096,-110.686,166.262,55.698,160.107
C06325=1016.660,37.847,-110.671,166.258,55.706,160.108
C06326=1016.655,37.596,-110.657,166.256,55.715,160.110
C06327=1016.650,37.347,-110.641,166.254,55.723,160.111
C06328=1016.645,37.097,-110.627,166.251,55.731,160.111
C06329=1016.639,36.848,-110.612,166.249,55.739,160.112
C06330=1016.634,36.599,-110.597,166.247,55.747,160.114
C06331=1016.629,36.349,-110.583,166.243,55.756,160.114
C06332=1016.624,36.100,-110.569,166.241,55.763,160.115
C06333=1016.619,35.850,-110.554,166.239,55.772,160.116
C06334=1016.613,35.601,-110.540,166.236,55.780,160.117
C06335=1016.608,35.351,-110.525,166.234,55.788,160.118
C06336=1016.602,35.101,-110.510,166.231,55.797,160.119
C06337=1016.597,34.851,-110.496,166.229,55.805,160.121
C06338=1016.592,34.602,-110.481,166.226,55.814,160.122
C06339=1016.587,34.352,-110.467,166.223,55.822,160.122
C06340=1016.581,34.103,-110.452,166.221,55.830,160.123
C06341=1016.576,33.854,-110.438,166.218,55.838,160.124
C06342=1016.571,33.604,-110.424,166.216,55.847,160.125
C06343=1016.566,33.355,-110.409,166.214,55.855,160.127
C06344=1016.560,33.105,-110.395,166.210,55.863,160.127
C06345=1016.556,32.855,-110.380,166.208,55.871,160.128
C06346=1016.550,32.606,-110.366,166.206,55.879,160.129
C06347=1016.545,32.356,-110.351,166.203,55.888,160.130
C06348=1016.540,32.107,-110.338,166.201,55.896,160.132
C06349=1016.535,31.858,-110.322,166.198,55.904,160.132
C06350=1016.529,31.608,-110.309,166.195,55.912,160.133
C06351=1016.524,31.358,-110.295,166.193,55.921,160.134
C06352=1016.519,31.109,-110.279,166.190,55.929,160.135
C06353=1016.513,30.860,-110.266,166.187,55.937,160.136
C06354=1016.508,30.610,-110.251,166.185,55.945,160.137
C06355=1016.503,30.361,-110.237,166.182,55.954,160.138
C06356=1016.498,30.111,-110.222,166.180,55.961,160.139
C06357=1016.492,29.861,-110.208,166.178,55.970,160.140
C06358=1016.487,29.612,-110.193,166.175,55.978,160.141
C06359=1016.482,29.362,-110.179,166.172,55.986,160.142
C06360=1016.477,29.113,-110.165,166.170,55.994,160.143
C06361=1016.472,28.863,-110.151,166.167,56.003,160.144
C06362=1016.467,28.614,-110.136,166.165,56.010,160.145
C06363=1016.461,28.364,-110.122,166.163,56.019,160.146
C06364=1016.456,28.114,-110.107,166.161,56.027,160.147
C06365=1016.451,27.865,-110.094,166.157,56.035,160.148
C06366=1016.446,27.615,-110.079,166.155,56.043,160.149
C06367=1016.440,27.366,-110.064,166.153,56.051,160.150
C06368=1016.435,27.116,-110.051,166.149,56.059,160.151
C06369=1016.429,26.834,-110.035,166.147,56.069,160.152
C06370=1016.424,26.552,-110.018,166.144,56.078,160.153
C06371=1016.418,26.270,-110.002,166.142,56.088,160.154
C06372=1016.412,25.988,-109.987,166.138,56.097,160.155
C06373=1016.407,25.739,-109.973,166.136,56.105,160.156
C06374=1016.402,25.490,-109.959,166.134,56.113,160.157
C06375=1016.397,25.241,-109.944,166.130,56.121,160.158
C06376=1016.391,24.991,-109.930,166.128,56.130,160.159
C06377=1016.386,24.742,-109.917,166.125,56.138,160.160
C06378=1016.380,24.492,-109.903,166.123,56.147,160.161
C06379=1016.375,24.242,-109.889,166.121,56.154,160.162
C06380=1016.370,23.992,-109.874,166.118,56.163,160.163
C06381=1016.364,23.743,-109.861,166.116,56.171,160.164
C06382=1016.359,23.493,-109.847,166.113,56.179,160.165
C06383=1016.354,23.244,-109.833,166.110,56.187,160.166
C06384=1016.349,22.995,-109.819,166.108,56.196,160.167
C06385=1016.344,22.745,-109.805,166.106,56.203,160.168
C06386=1016.338,22.495,-109.791,166.103,56.212,160.169
C06387=1016.333,22.246,-109.777,166.101,56.220,160.170
C06388=1016.327,21.996,-109.763,166.097,56.228,160.171
C06389=1016.323,21.746,-109.749,166.095,56.237,160.172
C06390=1016.318,21.498,-109.735,166.093,56.244,160.173
C06391=1016.312,21.248,-109.721,166.090,56.253,160.174
C06392=1016.307,20.998,-109.708,166.088,56.261,160.175
C06393=1016.302,20.748,-109.693,166.085,56.269,160.176
C06394=1016.297,20.498,-109.680,166.082,56.277,160.177
C06395=1016.291,20.249,-109.666,166.080,56.285,160.177
C06396=1016.287,20.000,-109.653,166.078,56.293,160.179
C06397=1016.281,19.750,-109.639,166.075,56.302,160.180
C06398=1016.276,19.500,-109.624,166.072,56.310,160.180
C06399=1016.271,19.251,-109.610,166.070,56.318,160.182
C06400=1016.265,19.001,-109.597,166.067,56.326,160.182
C06401=1016.260,18.752,-109.583,166.065,56.334,160.183
C06402=1016.255,18.503,-109.569,166.062,56.342,160.184
C06403=1016.250,18.253,-109.555,166.059,56.351,160.185
C06404=1016.244,18.003,-109.542,166.057,56.359,160.186
C06405=1016.239,17.753,-109.528,166.055,56.366,160.187
C06406=1016.233,17.504,-109.514,166.052,56.375,160.188
C06407=1016.229,17.255,-109.500,166.050,56.383,160.189
C06408=1016.224,17.005,-109.486,166.046,56.391,160.190
C06409=1016.219,16.755,-109.473,166.044,56.400,160.191
C06410=1016.213,16.505,-109.459,166.042,56.407,160.192
C06411=1016.208,16.256,-109.446,166.039,56.416,160.193
C06412=1016.203,16.007,-109.432,166.037,56.424,160.194
C06413=1016.198,15.757,-109.419,166.035,56.432,160.195
C06414=1016.192,15.507,-109.405,166.031,56.440,160.195
C06415=1016.187,15.258,-109.392,166.029,56.448,160.197
C06416=1016.182,15.009,-109.378,166.027,56.457,160.198
C06417=1016.177,14.758,-109.365,166.024,56.465,160.198
C06418=1016.171,14.509,-109.351,166.022,56.473,160.200
C06419=1016.166,14.260,-109.337,166.019,56.481,160.200
C06420=1016.161,14.010,-109.323,166.016,56.489,160.201
C06421=1016.156,13.760,-109.310,166.014,56.497,160.202
C06422=1016.150,13.511,-109.296,166.011,56.505,160.203
C06423=1016.146,13.261,-109.283,166.008,56.513,160.204
C06424=1016.141,13.011,-109.269,166.006,56.521,160.205
C06425=1016.135,12.762,-109.256,166.004,56.529,160.206
C06426=1016.130,12.512,-109.243,166.001,56.538,160.207
C06427=1016.125,12.263,-109.229,165.999,56.546,160.208
C06428=1016.119,12.013,-109.216,165.996,56.554,160.209
C06429=1016.113,11.763,-109.203,165.994,56.563,160.210
C06430=1016.109,11.514,-109.190,165.990,56.571,160.211
C06431=1016.103,11.264,-109.176,165.988,56.579,160.212
C06432=1016.098,11.014,-109.163,165.987,56.588,160.213
C06433=1016.092,10.735,-109.148,165.983,56.597,160.214
C06434=1016.086,10.454,-109.133,165.980,56.606,160.215
C06435=1016.080,10.173,-109.118,165.977,56.615,160.216
C06436=1016.075,9.893,-109.104,165.975,56.624,160.217
C06437=1016.068,9.644,-109.090,165.971,56.632,160.218
C06438=1016.064,9.394,-109.078,165.969,56.641,160.219
C06439=1016.058,9.144,-109.064,165.966,56.649,160.220
C06440=1016.053,8.894,-109.051,165.964,56.657,160.221
C06441=1016.048,8.646,-109.038,165.962,56.665,160.222
C06442=1016.042,8.396,-109.025,165.959,56.674,160.223
C06443=1016.037,8.146,-109.011,165.956,56.681,160.223
C06444=1016.032,7.896,-108.998,165.954,56.690,160.225
C06445=1016.026,7.647,-108.985,165.951,56.698,160.225
C06446=1016.021,7.397,-108.971,165.949,56.706,160.226
C06447=1016.016,7.147,-108.959,165.946,56.714,160.227
C06448=1016.011,6.898,-108.945,165.944,56.722,160.228
C06449=1016.006,6.649,-108.933,165.941,56.730,160.229
C06450=1016.000,6.399,-108.919,165.938,56.739,160.230
C06451=1015.995,6.149,-108.906,165.936,56.747,160.231
C06452=1015.990,5.899,-108.893,165.934,56.755,160.232
C06453=1015.985,5.650,-108.879,165.931,56.763,160.233
C06454=1015.980,5.401,-108.867,165.928,56.771,160.234
C06455=1015.974,5.151,-108.854,165.926,56.779,160.235
C06456=1015.969,4.901,-108.840,165.923,56.787,160.235
C06457=1015.964,4.651,-108.827,165.921,56.795,160.237
C06458=1015.958,4.402,-108.814,165.919,56.803,160.237
C06459=1015.954,4.153,-108.801,165.915,56.811,160.238
C06460=1015.948,3.903,-108.788,165.913,56.819,160.239
C06461=1015.944,3.653,-108.775,165.911,56.827,160.240
C06462=1015.938,3.404,-108.762,165.907,56.835,160.241
C06463=1015.933,3.154,-108.749,165.906,56.844,160.242
C06464=1015.928,2.904,-108.736,165.903,56.851,160.243
C06465=1015.922,2.654,-108.722,165.900,56.859,160.244
C06466=1015.917,2.405,-108.710,165.898,56.868,160.245
C06467=1015.912,2.155,-108.697,165.896,56.875,160.246
C06468=1015.907,1.906,-108.683,165.892,56.883,160.246
C06469=1015.902,1.656,-108.670,165.890,56.892,160.247
C06470=1015.897,1.407,-108.658,165.888,56.899,160.248
C06471=1015.891,1.157,-108.645,165.884,56.908,160.249
C06472=1015.887,0.908,-108.631,165.882,56.915,160.250
C06473=1015.881,0.658,-108.618,165.880,56.924,160.251
C06474=1015.876,0.408,-108.606,165.878,56.931,160.252
C06475=1015.871,0.158,-108.593,165.874,56.939,160.252
C06476=1015.866,-0.091,-108.579,165.872,56.947,160.253
C06477=1015.861,-0.341,-108.566,165.870,56.955,160.255
C06478=1015.856,-0.590,-108.554,165.868,56.963,160.255
C06479=1015.850,-0.840,-108.541,165.864,56.971,160.256
C06480=1015.846,-1.090,-108.528,165.862,56.979,160.257
C06481=1015.840,-1.339,-108.514,165.860,56.986,160.258
C06482=1015.835,-1.588,-108.502,165.858,56.995,160.259
C06483=1015.830,-1.838,-108.489,165.854,57.003,160.260
C06484=1015.825,-2.088,-108.476,165.852,57.011,160.261
C06485=1015.820,-2.337,-108.464,165.850,57.018,160.261
C06486=1015.814,-2.587,-108.450,165.847,57.026,160.262
C06487=1015.810,-2.836,-108.437,165.844,57.034,160.263
C06488=1015.805,-3.087,-108.424,165.841,57.042,160.264
C06489=1015.799,-3.336,-108.412,165.839,57.049,160.265
C06490=1015.794,-3.586,-108.399,165.837,57.058,160.266
C06491=1015.790,-3.835,-108.386,165.834,57.066,160.267
C06492=1015.785,-4.084,-108.372,165.831,57.074,160.267
C06493=1015.779,-4.334,-108.360,165.829,57.081,160.268
C06494=1015.774,-4.584,-108.347,165.827,57.089,160.269
C06495=1015.768,-4.834,-108.334,165.823,57.097,160.270
C06496=1015.764,-5.084,-108.322,165.821,57.105,160.271
C06497=1015.758,-5.368,-108.307,165.819,57.114,160.272
C06498=1015.752,-5.653,-108.294,165.815,57.124,160.273
C06499=1015.746,-5.938,-108.279,165.812,57.133,160.274
C06500=1015.740,-6.222,-108.265,165.810,57.142,160.275
C06501=1015.734,-6.472,-108.252,165.807,57.150,160.276
C06502=1015.729,-6.722,-108.240,165.804,57.159,160.277
C06503=1015.724,-6.971,-108.227,165.802,57.166,160.278
C06504=1015.719,-7.222,-108.215,165.799,57.174,160.278
C06505=1015.713,-7.471,-108.203,165.796,57.182,160.279
C06506=1015.709,-7.720,-108.190,165.795,57.190,160.280
C06507=1015.703,-7.970,-108.178,165.791,57.199,160.281
C06508=1015.698,-8.220,-108.165,165.789,57.206,160.282
C06509=1015.693,-8.469,-108.153,165.786,57.214,160.283
C06510=1015.687,-8.719,-108.140,165.783,57.222,160.283
C06511=1015.683,-8.969,-108.128,165.781,57.230,160.285
C06512=1015.678,-9.218,-108.116,165.779,57.238,160.286
C06513=1015.672,-9.468,-108.104,165.776,57.246,160.286
C06514=1015.667,-9.717,-108.091,165.773,57.254,160.287
C06515=1015.662,-9.966,-108.079,165.771,57.262,160.288
C06516=1015.656,-10.217,-108.067,165.769,57.269,160.289
C06517=1015.652,-10.466,-108.054,165.765,57.278,160.289
C06518=1015.646,-10.716,-108.042,165.763,57.286,160.291
C06519=1015.641,-10.966,-108.029,165.761,57.294,160.292
C06520=1015.636,-11.215,-108.016,165.758,57.302,160.292
C06521=1015.631,-11.465,-108.005,165.755,57.310,160.293
C06522=1015.626,-11.715,-107.992,165.753,57.317,160.294
C06523=1015.620,-11.964,-107.980,165.751,57.325,160.295
C06524=1015.615,-12.213,-107.967,165.747,57.333,160.296
C06525=1015.611,-12.464,-107.955,165.745,57.341,160.296
C06526=1015.605,-12.713,-107.943,165.743,57.348,160.297
C06527=1015.600,-12.963,-107.931,165.739,57.357,160.298
C06528=1015.595,-13.212,-107.918,165.737,57.364,160.299
C06529=1015.590,-13.462,-107.906,165.735,57.372,160.300
C06530=1015.584,-13.712,-107.894,165.732,57.380,160.301
C06531=1015.580,-13.961,-107.881,165.729,57.388,160.301
C06532=1015.575,-14.211,-107.870,165.727,57.396,160.302
C06533=1015.570,-14.461,-107.857,165.724,57.403,160.303
C06534=1015.564,-14.710,-107.844,165.722,57.411,160.304
C06535=1015.559,-14.960,-107.833,165.720,57.419,160.305
C06536=1015.555,-15.210,-107.820,165.716,57.427,160.305
C06537=1015.549,-15.459,-107.808,165.714,57.435,160.306
C06538=1015.544,-15.709,-107.796,165.712,57.442,160.307
C06539=1015.539,-15.959,-107.783,165.710,57.450,160.308
C06540=1015.534,-16.208,-107.771,165.706,57.458,160.309
C06541=1015.529,-16.458,-107.760,165.704,57.466,160.310
C06542=1015.523,-16.708,-107.747,165.702,57.474,160.311
C06543=1015.518,-16.958,-107.736,165.698,57.482,160.311
C06544=1015.513,-17.207,-107.723,165.696,57.490,160.312
C06545=1015.508,-17.457,-107.712,165.694,57.497,160.313
C06546=1015.503,-17.706,-107.700,165.690,57.505,160.314
C06547=1015.497,-17.957,-107.687,165.689,57.514,160.315
C06548=1015.492,-18.206,-107.676,165.686,57.522,160.316
C06549=1015.487,-18.456,-107.664,165.683,57.530,160.316
C06550=1015.482,-18.705,-107.652,165.681,57.538,160.317
C06551=1015.477,-18.955,-107.640,165.678,57.545,160.318
C06552=1015.472,-19.204,-107.628,165.676,57.553,160.319
C06553=1015.467,-19.451,-107.617,165.673,57.561,160.320
C06554=1015.461,-19.697,-107.605,165.670,57.568,160.320
C06555=1015.456,-19.944,-107.593,165.668,57.576,160.321
C06556=1015.451,-20.190,-107.582,165.665,57.584,160.322
C06557=1015.446,-20.436,-107.570,165.663,57.591,160.323
C06558=1015.441,-20.683,-107.558,165.660,57.600,160.324
C06559=1015.436,-20.930,-107.546,165.657,57.607,160.325
C06560=1015.431,-21.175,-107.534,165.655,57.615,160.325
C06561=1015.425,-21.452,-107.522,165.652,57.623,160.326
C06562=1015.420,-21.729,-107.508,165.649,57.632,160.327
C06563=1015.414,-22.005,-107.495,165.646,57.641,160.328
C06564=1015.408,-22.282,-107.483,165.643,57.649,160.329
C06565=1015.404,-22.532,-107.471,165.641,57.657,160.330
C06566=1015.398,-22.781,-107.459,165.639,57.665,160.331
C06567=1015.393,-23.031,-107.447,165.636,57.673,160.331
C06568=1015.388,-23.281,-107.435,165.633,57.681,160.332
C06569=1015.382,-23.530,-107.423,165.631,57.688,160.333
C06570=1015.377,-23.780,-107.412,165.628,57.695,160.334
C06571=1015.372,-24.030,-107.400,165.626,57.703,160.334
C06572=1015.367,-24.279,-107.388,165.623,57.711,160.335
C06573=1015.362,-24.529,-107.376,165.620,57.719,160.336
C06574=1015.357,-24.779,-107.365,165.618,57.727,160.337
C06575=1015.352,-25.028,-107.353,165.615,57.734,160.337
C06576=1015.347,-25.278,-107.341,165.613,57.742,160.338
C06577=1015.342,-25.528,-107.330,165.610,57.749,160.339
C06578=1015.337,-25.777,-107.318,165.607,57.758,160.340
C06579=1015.331,-26.027,-107.306,165.604,57.765,160.341
C06580=1015.326,-26.276,-107.295,165.602,57.772,160.341
C06581=1015.321,-26.526,-107.283,165.600,57.780,160.342
C06582=1015.317,-26.776,-107.271,165.598,57.788,160.343
C06583=1015.312,-27.025,-107.259,165.595,57.795,160.344
C06584=1015.307,-27.275,-107.247,165.591,57.803,160.344
C06585=1015.302,-27.525,-107.236,165.589,57.811,160.345
C06586=1015.297,-27.775,-107.225,165.586,57.818,160.346
C06587=1015.292,-28.025,-107.213,165.584,57.826,160.347
C06588=1015.286,-28.274,-107.202,165.582,57.834,160.348
C06589=1015.281,-28.524,-107.191,165.579,57.842,160.348
C06590=1015.276,-28.773,-107.179,165.576,57.850,160.349
C06591=1015.271,-29.023,-107.167,165.573,57.857,160.350
C06592=1015.266,-29.273,-107.156,165.570,57.865,160.351
C06593=1015.260,-29.522,-107.145,165.568,57.873,160.351
C06594=1015.255,-29.772,-107.133,165.566,57.880,160.352
C06595=1015.250,-30.022,-107.122,165.564,57.888,160.353
C06596=1015.245,-30.272,-107.110,165.560,57.896,160.354
C06597=1015.239,-30.521,-107.099,165.557,57.903,160.355
C06598=1015.234,-30.771,-107.088,165.555,57.911,160.355
C06599=1015.229,-31.021,-107.076,165.553,57.919,160.356
C06600=1015.224,-31.270,-107.065,165.551,57.927,160.357
C06601=1015.219,-31.520,-107.054,165.547,57.934,160.358
C06602=1015.214,-31.770,-107.043,165.545,57.942,160.358
C06603=1015.209,-32.020,-107.031,165.542,57.950,160.359
C06604=1015.204,-32.269,-107.021,165.540,57.957,160.360
C06605=1015.199,-32.519,-107.009,165.536,57.965,160.361
C06606=1015.194,-32.769,-106.998,165.534,57.973,160.362
C06607=1015.189,-33.018,-106.987,165.532,57.981,160.362
C06608=1015.184,-33.268,-106.975,165.529,57.988,160.363
C06609=1015.179,-33.518,-106.964,165.527,57.995,160.364
C06610=1015.173,-33.767,-106.953,165.524,58.003,160.364
C06611=1015.168,-34.017,-106.942,165.521,58.011,160.365
C06612=1015.163,-34.267,-106.930,165.519,58.019,160.366
C06613=1015.159,-34.516,-106.919,165.516,58.026,160.367
C06614=1015.153,-34.766,-106.908,165.514,58.033,160.368
C06615=1015.148,-35.015,-106.897,165.511,58.041,160.368
C06616=1015.143,-35.266,-106.886,165.509,58.048,160.369
C06617=1015.138,-35.516,-106.874,165.505,58.056,160.370
C06618=1015.132,-35.765,-106.864,165.503,58.064,160.370
C06619=1015.127,-36.015,-106.852,165.500,58.071,160.371
C06620=1015.123,-36.264,-106.841,165.498,58.078,160.372
C06621=1015.118,-36.514,-106.830,165.495,58.086,160.373
C06622=1015.112,-36.763,-106.819,165.493,58.093,160.373
C06623=1015.108,-37.014,-106.808,165.490,58.101,160.374
C06624=1015.103,-37.264,-106.796,165.488,58.108,160.375
C06625=1015.097,-37.538,-106.784,165.485,58.117,160.376
C06626=1015.091,-37.813,-106.772,165.482,58.125,160.376
C06627=1015.087,-38.090,-106.760,165.478,58.134,160.377
C06628=1015.081,-38.365,-106.747,165.476,58.141,160.378
C06629=1015.075,-38.614,-106.736,165.473,58.148,160.379
C06630=1015.070,-38.865,-106.725,165.471,58.156,160.379
C06631=1015.066,-39.114,-106.714,165.467,58.164,160.380
C06632=1015.061,-39.364,-106.703,165.465,58.172,160.381
C06633=1015.055,-39.613,-106.692,165.462,58.179,160.381
C06634=1015.050,-39.864,-106.681,165.460,58.186,160.382
C06635=1015.045,-40.112,-106.671,165.458,58.194,160.383
C06636=1015.041,-40.363,-106.660,165.455,58.201,160.384
C06637=1015.035,-40.612,-106.649,165.453,58.208,160.384
C06638=1015.030,-40.862,-106.638,165.449,58.217,160.385
C06639=1015.025,-41.112,-106.628,165.447,58.225,160.386
C06640=1015.020,-41.361,-106.616,165.444,58.232,160.386
C06641=1015.015,-41.611,-106.606,165.442,58.239,160.387
C06642=1015.010,-41.861,-106.595,165.439,58.247,160.388
C06643=1015.005,-42.111,-106.585,165.437,58.254,160.389
C06644=1015.000,-42.360,-106.573,165.433,58.262,160.389
C06645=1014.994,-42.610,-106.563,165.431,58.270,160.390
C06646=1014.989,-42.860,-106.552,165.429,58.277,160.391
C06647=1014.984,-43.109,-106.541,165.426,58.284,160.391
C06648=1014.980,-43.360,-106.531,165.424,58.292,160.392
C06649=1014.974,-43.609,-106.520,165.421,58.299,160.393
C06650=1014.970,-43.859,-106.509,165.419,58.307,160.394
C06651=1014.964,-44.108,-106.498,165.416,58.314,160.394
C06652=1014.959,-44.358,-106.488,165.414,58.322,160.395
C06653=1014.954,-44.607,-106.477,165.410,58.329,160.396
C06654=1014.949,-44.858,-106.467,165.407,58.336,160.396
C06655=1014.944,-45.107,-106.455,165.405,58.344,160.397
C06656=1014.939,-45.357,-106.446,165.402,58.351,160.398
C06657=1014.934,-45.607,-106.434,165.400,58.358,160.398
C06658=1014.928,-45.857,-106.424,165.397,58.366,160.399
///RCONF 1,0,0,1,0,0,0,0,0,0,0,0,0,0,0,0,0,0,0,0,0,0,0,0
C06659=1014.924,-46.106,-106.413,165.395,58.373,160.400
C06660=1014.919,-46.356,-106.403,165.392,58.380,160.400
C06661=1014.914,-46.606,-106.392,165.390,58.388,160.401
C06662=1014.909,-46.855,-106.382,165.387,58.395,160.402
C06663=1014.904,-47.106,-106.371,165.384,58.402,160.402
C06664=1014.899,-47.354,-106.360,165.382,58.410,160.403
C06665=1014.894,-47.605,-106.350,165.379,58.417,160.404
C06666=1014.888,-47.854,-106.339,165.377,58.424,160.404
C06667=1014.884,-48.104,-106.328,165.374,58.431,160.405
C06668=1014.879,-48.354,-106.318,165.372,58.439,160.406
C06669=1014.874,-48.603,-106.308,165.369,58.446,160.407
C06670=1014.869,-48.853,-106.297,165.366,58.453,160.407
C06671=1014.864,-49.103,-106.287,165.363,58.461,160.408
C06672=1014.859,-49.352,-106.276,165.361,58.468,160.408
C06673=1014.854,-49.603,-106.265,165.359,58.475,160.409
C06674=1014.849,-49.852,-106.254,165.356,58.483,160.410
C06675=1014.844,-50.102,-106.244,165.353,58.490,160.410
C06676=1014.840,-50.352,-106.234,165.350,58.497,160.411
C06677=1014.834,-50.602,-106.224,165.348,58.504,160.412
C06678=1014.829,-50.851,-106.212,165.345,58.511,160.412
C06679=1014.825,-51.101,-106.202,165.342,58.518,160.413
C06680=1014.819,-51.351,-106.192,165.340,58.526,160.414
C06681=1014.814,-51.600,-106.182,165.337,58.533,160.414
C06682=1014.810,-51.851,-106.172,165.335,58.541,160.415
C06683=1014.805,-52.100,-106.162,165.331,58.549,160.415
C06684=1014.799,-52.350,-106.152,165.329,58.556,160.416
C06685=1014.794,-52.599,-106.141,165.327,58.563,160.417
C06686=1014.789,-52.849,-106.131,165.324,58.571,160.418
C06687=1014.784,-53.099,-106.121,165.321,58.578,160.418
C06688=1014.779,-53.349,-106.111,165.319,58.586,160.419
C06689=1014.773,-53.625,-106.101,165.316,58.594,160.420
C06690=1014.768,-53.900,-106.089,165.313,58.602,160.420
C06691=1014.761,-54.176,-106.078,165.311,58.610,160.421
C06692=1014.756,-54.452,-106.067,165.307,58.618,160.422
C06693=1014.751,-54.702,-106.057,165.305,58.625,160.423
C06694=1014.746,-54.952,-106.047,165.302,58.633,160.423
C06695=1014.741,-55.201,-106.037,165.299,58.640,160.424
C06696=1014.736,-55.451,-106.027,165.296,58.647,160.424
C06697=1014.731,-55.701,-106.017,165.294,58.655,160.425
C06698=1014.726,-55.950,-106.007,165.291,58.662,160.426
C06699=1014.721,-56.200,-105.997,165.288,58.669,160.426
C06700=1014.716,-56.450,-105.988,165.285,58.677,160.427
C06701=1014.710,-56.700,-105.977,165.282,58.684,160.427
C06702=1014.705,-56.949,-105.968,165.280,58.692,160.428
C06703=1014.701,-57.198,-105.958,165.278,58.699,160.429
C06704=1014.695,-57.449,-105.948,165.275,58.706,160.430
C06705=1014.690,-57.698,-105.938,165.272,58.713,160.430
C06706=1014.685,-57.948,-105.928,165.270,58.720,160.431
C06707=1014.681,-58.198,-105.917,165.267,58.727,160.431
C06708=1014.676,-58.447,-105.907,165.264,58.734,160.432
C06709=1014.671,-58.698,-105.898,165.261,58.742,160.432
C06710=1014.666,-58.947,-105.888,165.259,58.749,160.433
C06711=1014.661,-59.197,-105.878,165.257,58.757,160.434
C06712=1014.656,-59.447,-105.868,165.254,58.764,160.435
C06713=1014.651,-59.696,-105.858,165.251,58.771,160.435
C06714=1014.645,-59.946,-105.848,165.249,58.778,160.436
C06715=1014.641,-60.196,-105.839,165.247,58.785,160.437
C06716=1014.636,-60.445,-105.829,165.244,58.792,160.437
C06717=1014.631,-60.696,-105.819,165.242,58.799,160.438
C06718=1014.626,-60.945,-105.809,165.239,58.806,160.438
C06719=1014.621,-61.195,-105.800,165.236,58.813,160.439
C06720=1014.616,-61.445,-105.790,165.233,58.820,160.439
C06721=1014.611,-61.694,-105.780,165.231,58.828,160.440
C06722=1014.606,-61.944,-105.770,165.228,58.835,160.441
C06723=1014.601,-62.194,-105.760,165.225,58.841,160.441
C06724=1014.596,-62.444,-105.751,165.222,58.848,160.442
C06725=1014.591,-62.693,-105.741,165.219,58.855,160.442
C06726=1014.586,-62.943,-105.731,165.218,58.862,160.443
C06727=1014.581,-63.193,-105.721,165.215,58.869,160.444
C06728=1014.576,-63.443,-105.712,165.212,58.876,160.444
C06729=1014.571,-63.692,-105.702,165.210,58.884,160.445
C06730=1014.566,-63.942,-105.692,165.207,58.891,160.445
C06731=1014.561,-64.192,-105.682,165.204,58.897,160.446
C06732=1014.557,-64.442,-105.673,165.201,58.904,160.446
C06733=1014.551,-64.692,-105.663,165.199,58.911,160.447
C06734=1014.546,-64.941,-105.653,165.197,58.918,160.448
C06735=1014.542,-65.191,-105.643,165.194,58.925,160.448
C06736=1014.537,-65.441,-105.634,165.191,58.932,160.448
C06737=1014.532,-65.691,-105.624,165.188,58.939,160.449
C06738=1014.527,-65.940,-105.614,165.186,58.946,160.450
C06739=1014.523,-66.191,-105.605,165.184,58.953,160.450
C06740=1014.518,-66.440,-105.595,165.180,58.959,160.451
C06741=1014.513,-66.689,-105.585,165.178,58.966,160.451
C06742=1014.508,-66.939,-105.575,165.175,58.973,160.452
C06743=1014.503,-67.189,-105.566,165.173,58.979,160.452
C06744=1014.499,-67.439,-105.556,165.170,58.987,160.453
C06745=1014.494,-67.688,-105.546,165.168,58.994,160.453
C06746=1014.489,-67.938,-105.537,165.164,59.000,160.454
C06747=1014.484,-68.188,-105.527,165.163,59.007,160.455
C06748=1014.479,-68.438,-105.518,165.160,59.014,160.455
C06749=1014.474,-68.688,-105.508,165.157,59.021,160.455
C06750=1014.470,-68.937,-105.498,165.154,59.028,160.456
C06751=1014.465,-69.187,-105.489,165.152,59.034,160.457
C06752=1014.460,-69.437,-105.479,165.149,59.041,160.457
C06753=1014.454,-69.714,-105.468,165.146,59.048,160.458
C06754=1014.449,-69.991,-105.458,165.143,59.056,160.458
C06755=1014.443,-70.267,-105.447,165.141,59.064,160.459
C06756=1014.439,-70.544,-105.437,165.138,59.071,160.460
C06757=1014.434,-70.794,-105.427,165.135,59.077,160.460
C06758=1014.429,-71.044,-105.418,165.132,59.084,160.460
C06759=1014.424,-71.293,-105.408,165.130,59.090,160.461
C06760=1014.420,-71.543,-105.399,165.127,59.097,160.461
C06761=1014.415,-71.793,-105.389,165.125,59.103,160.462
C06762=1014.410,-72.042,-105.379,165.122,59.111,160.463
C06763=1014.406,-72.292,-105.370,165.119,59.117,160.463
C06764=1014.400,-72.542,-105.360,165.117,59.124,160.464
C06765=1014.396,-72.792,-105.351,165.114,59.130,160.464
C06766=1014.391,-73.042,-105.341,165.111,59.137,160.464
C06767=1014.386,-73.292,-105.332,165.109,59.143,160.465
C06768=1014.381,-73.541,-105.323,165.106,59.150,160.465
C06769=1014.377,-73.791,-105.313,165.104,59.157,160.466
C06770=1014.372,-74.041,-105.304,165.101,59.163,160.466
C06771=1014.368,-74.291,-105.295,165.098,59.169,160.467
C06772=1014.363,-74.540,-105.285,165.096,59.176,160.467
C06773=1014.358,-74.790,-105.276,165.093,59.183,160.468
C06774=1014.353,-75.040,-105.267,165.091,59.189,160.468
C06775=1014.348,-75.289,-105.257,165.088,59.196,160.469
C06776=1014.344,-75.539,-105.248,165.085,59.203,160.469
C06777=1014.339,-75.789,-105.239,165.082,59.209,160.470
C06778=1014.334,-76.039,-105.231,165.081,59.216,160.470
C06779=1014.329,-76.288,-105.221,165.077,59.223,160.471
C06780=1014.324,-76.538,-105.212,165.075,59.230,160.471
C06781=1014.319,-76.788,-105.203,165.072,59.236,160.472
C06782=1014.315,-77.038,-105.194,165.070,59.243,160.472
C06783=1014.310,-77.287,-105.185,165.067,59.249,160.473
C06784=1014.305,-77.537,-105.176,165.065,59.256,160.473
C06785=1014.300,-77.787,-105.167,165.062,59.263,160.474
C06786=1014.296,-78.037,-105.158,165.060,59.269,160.474
C06787=1014.291,-78.287,-105.148,165.057,59.276,160.475
C06788=1014.285,-78.536,-105.140,165.054,59.282,160.475
C06789=1014.281,-78.786,-105.131,165.052,59.289,160.476
C06790=1014.276,-79.036,-105.121,165.049,59.295,160.476
C06791=1014.271,-79.286,-105.113,165.046,59.302,160.476
C06792=1014.266,-79.536,-105.103,165.044,59.309,160.477
C06793=1014.262,-79.786,-105.094,165.041,59.315,160.477
C06794=1014.256,-80.035,-105.086,165.039,59.321,160.478
C06795=1014.252,-80.285,-105.077,165.036,59.328,160.479
C06796=1014.247,-80.535,-105.067,165.034,59.334,160.479
C06797=1014.242,-80.785,-105.059,165.030,59.341,160.479
C06798=1014.238,-81.035,-105.050,165.028,59.348,160.480
C06799=1014.232,-81.285,-105.041,165.026,59.354,160.480
C06800=1014.228,-81.535,-105.032,165.023,59.361,160.481
C06801=1014.223,-81.785,-105.024,165.020,59.368,160.481
C06802=1014.217,-82.034,-105.015,165.018,59.374,160.482
C06803=1014.213,-82.284,-105.006,165.015,59.381,160.482
C06804=1014.208,-82.533,-104.998,165.012,59.387,160.483
C06805=1014.204,-82.783,-104.989,165.010,59.394,160.483
C06806=1014.198,-83.033,-104.981,165.007,59.401,160.484
C06807=1014.193,-83.283,-104.972,165.004,59.408,160.484
C06808=1014.189,-83.533,-104.963,165.002,59.414,160.485
C06809=1014.184,-83.783,-104.955,164.999,59.420,160.485
C06810=1014.179,-84.033,-104.946,164.997,59.427,160.486
C06811=1014.174,-84.282,-104.938,164.994,59.434,160.486
C06812=1014.170,-84.532,-104.929,164.992,59.440,160.487
C06813=1014.165,-84.782,-104.920,164.989,59.446,160.487
C06814=1014.159,-85.032,-104.912,164.986,59.453,160.487
C06815=1014.155,-85.282,-104.903,164.984,59.459,160.488
C06816=1014.150,-85.531,-104.894,164.980,59.466,160.488
C06817=1014.145,-85.810,-104.885,164.978,59.473,160.489
C06818=1014.139,-86.089,-104.875,164.975,59.480,160.489
C06819=1014.134,-86.368,-104.867,164.973,59.487,160.490
C06820=1014.129,-86.646,-104.857,164.969,59.494,160.490
C06821=1014.123,-86.896,-104.848,164.967,59.501,160.491
C06822=1014.119,-87.145,-104.839,164.965,59.507,160.491
C06823=1014.114,-87.395,-104.831,164.961,59.514,160.491
C06824=1014.110,-87.646,-104.822,164.959,59.520,160.492
C06825=1014.105,-87.895,-104.814,164.956,59.526,160.492
C06826=1014.099,-88.145,-104.806,164.954,59.532,160.493
C06827=1014.095,-88.394,-104.797,164.951,59.539,160.493
C06828=1014.090,-88.644,-104.788,164.948,59.545,160.493
C06829=1014.086,-88.895,-104.780,164.946,59.552,160.494
C06830=1014.081,-89.144,-104.771,164.944,59.558,160.495
C06831=1014.076,-89.393,-104.763,164.941,59.564,160.495
C06832=1014.071,-89.644,-104.754,164.938,59.570,160.495
C06833=1014.067,-89.894,-104.747,164.936,59.576,160.496
C06834=1014.062,-90.144,-104.737,164.933,59.583,160.496
C06835=1014.057,-90.393,-104.729,164.931,59.589,160.496
C06836=1014.052,-90.643,-104.721,164.928,59.595,160.497
C06837=1014.048,-90.893,-104.712,164.925,59.601,160.497
C06838=1014.043,-91.142,-104.704,164.923,59.607,160.498
C06839=1014.039,-91.392,-104.695,164.920,59.614,160.498
C06840=1014.034,-91.643,-104.687,164.918,59.620,160.498
C06841=1014.029,-91.892,-104.679,164.915,59.626,160.499
C06842=1014.025,-92.142,-104.670,164.912,59.632,160.499
C06843=1014.020,-92.392,-104.663,164.909,59.638,160.499
C06844=1014.016,-92.641,-104.654,164.907,59.644,160.500
C06845=1014.010,-92.891,-104.645,164.904,59.650,160.500
C06846=1014.005,-93.141,-104.638,164.902,59.656,160.501
C06847=1014.001,-93.391,-104.629,164.900,59.662,160.501
C06848=1013.996,-93.640,-104.620,164.898,59.668,160.502
C06849=1013.992,-93.891,-104.612,164.894,59.674,160.501
C06850=1013.987,-94.140,-104.604,164.891,59.680,160.502
C06851=1013.982,-94.390,-104.595,164.889,59.686,160.502
C06852=1013.978,-94.640,-104.587,164.886,59.693,160.503
C06853=1013.973,-94.889,-104.579,164.884,59.699,160.503
C06854=1013.969,-95.139,-104.570,164.881,59.704,160.503
C06855=1013.964,-95.390,-104.562,164.879,59.710,160.504
C06856=1013.959,-95.639,-104.554,164.877,59.716,160.504
C06857=1013.955,-95.889,-104.546,164.874,59.723,160.505
C06858=1013.950,-96.138,-104.537,164.871,59.728,160.505
C06859=1013.945,-96.389,-104.530,164.869,59.734,160.505
C06860=1013.941,-96.639,-104.521,164.866,59.740,160.506
C06861=1013.936,-96.888,-104.512,164.864,59.745,160.506
C06862=1013.932,-97.139,-104.504,164.860,59.752,160.506
C06863=1013.927,-97.388,-104.496,164.858,59.758,160.507
C06864=1013.922,-97.638,-104.488,164.855,59.763,160.507
C06865=1013.918,-97.887,-104.480,164.853,59.769,160.507
C06866=1013.913,-98.138,-104.472,164.851,59.775,160.508
C06867=1013.908,-98.387,-104.463,164.847,59.781,160.508
C06868=1013.904,-98.637,-104.456,164.845,59.787,160.508
C06869=1013.899,-98.887,-104.448,164.843,59.793,160.509
C06870=1013.895,-99.137,-104.439,164.841,59.799,160.509
C06871=1013.890,-99.387,-104.432,164.837,59.805,160.509
C06872=1013.885,-99.636,-104.424,164.835,59.811,160.509
C06873=1013.880,-99.886,-104.416,164.833,59.817,160.510
C06874=1013.876,-100.136,-104.408,164.831,59.823,160.510
C06875=1013.871,-100.386,-104.401,164.828,59.828,160.511
C06876=1013.866,-100.635,-104.392,164.825,59.835,160.511
C06877=1013.861,-100.886,-104.385,164.822,59.841,160.511
C06878=1013.857,-101.135,-104.377,164.820,59.846,160.511
C06879=1013.852,-101.386,-104.369,164.817,59.852,160.512
C06880=1013.848,-101.635,-104.361,164.815,59.858,160.512
C06881=1013.843,-101.916,-104.353,164.812,59.865,160.513
C06882=1013.838,-102.196,-104.344,164.809,59.871,160.513
C06883=1013.832,-102.478,-104.334,164.806,59.878,160.513
C06884=1013.827,-102.758,-104.325,164.804,59.884,160.514
C06885=1013.823,-103.008,-104.318,164.800,59.890,160.514
C06886=1013.818,-103.258,-104.310,164.798,59.896,160.514
C06887=1013.813,-103.507,-104.302,164.795,59.902,160.515
C06888=1013.809,-103.757,-104.295,164.793,59.907,160.515
C06889=1013.804,-104.007,-104.287,164.790,59.913,160.515
C06890=1013.799,-104.257,-104.280,164.788,59.918,160.515
C06891=1013.794,-104.507,-104.272,164.786,59.924,160.516
C06892=1013.790,-104.756,-104.264,164.783,59.930,160.516
C06893=1013.785,-105.006,-104.256,164.781,59.936,160.516
C06894=1013.780,-105.256,-104.249,164.778,59.941,160.517
C06895=1013.776,-105.505,-104.241,164.776,59.947,160.517
C06896=1013.772,-105.756,-104.233,164.773,59.952,160.517
C06897=1013.767,-106.006,-104.225,164.771,59.959,160.518
C06898=1013.762,-106.256,-104.218,164.768,59.964,160.518
C06899=1013.758,-106.505,-104.209,164.766,59.970,160.518
C06900=1013.753,-106.755,-104.202,164.763,59.975,160.518
C06901=1013.748,-107.005,-104.194,164.760,59.981,160.519
C06902=1013.744,-107.255,-104.187,164.758,59.987,160.519
C06903=1013.740,-107.504,-104.180,164.755,59.992,160.519
C06904=1013.735,-107.755,-104.172,164.753,59.997,160.519
C06905=1013.730,-108.004,-104.164,164.750,60.003,160.520
C06906=1013.726,-108.254,-104.157,164.748,60.009,160.520
C06907=1013.721,-108.504,-104.149,164.746,60.015,160.521
C06908=1013.716,-108.754,-104.142,164.743,60.020,160.521
C06909=1013.712,-109.003,-104.135,164.740,60.025,160.521
C06910=1013.707,-109.254,-104.127,164.738,60.031,160.521
C06911=1013.702,-109.503,-104.120,164.735,60.037,160.521
C06912=1013.698,-109.753,-104.112,164.733,60.043,160.522
C06913=1013.693,-110.003,-104.105,164.730,60.048,160.522
C06914=1013.689,-110.253,-104.097,164.727,60.053,160.522
C06915=1013.684,-110.502,-104.090,164.725,60.059,160.522
C06916=1013.680,-110.752,-104.082,164.722,60.065,160.523
C06917=1013.674,-111.002,-104.075,164.720,60.070,160.523
C06918=1013.670,-111.252,-104.068,164.717,60.075,160.523
C06919=1013.666,-111.502,-104.061,164.715,60.081,160.524
C06920=1013.661,-111.752,-104.053,164.712,60.087,160.524
C06921=1013.656,-112.002,-104.046,164.709,60.092,160.524
C06922=1013.652,-112.252,-104.039,164.706,60.097,160.524
C06923=1013.648,-112.501,-104.031,164.705,60.102,160.524
C06924=1013.643,-112.752,-104.023,164.703,60.108,160.525
C06925=1013.638,-113.001,-104.016,164.700,60.114,160.525
C06926=1013.633,-113.251,-104.009,164.697,60.119,160.525
C06927=1013.629,-113.501,-104.002,164.694,60.124,160.525
C06928=1013.624,-113.751,-103.995,164.692,60.130,160.525
C06929=1013.620,-114.001,-103.987,164.690,60.135,160.526
C06930=1013.616,-114.250,-103.980,164.687,60.140,160.526
C06931=1013.611,-114.500,-103.973,164.685,60.146,160.526
C06932=1013.607,-114.750,-103.965,164.682,60.151,160.527
C06933=1013.602,-115.001,-103.958,164.679,60.157,160.527
C06934=1013.597,-115.250,-103.951,164.678,60.161,160.527
C06935=1013.593,-115.500,-103.944,164.675,60.167,160.527
C06936=1013.588,-115.749,-103.936,164.672,60.172,160.527
C06937=1013.584,-115.999,-103.930,164.669,60.177,160.528
C06938=1013.579,-116.249,-103.923,164.667,60.183,160.528
C06939=1013.574,-116.499,-103.915,164.665,60.188,160.528
C06940=1013.570,-116.749,-103.908,164.662,60.193,160.528
C06941=1013.566,-116.999,-103.901,164.659,60.198,160.528
C06942=1013.561,-117.248,-103.894,164.657,60.204,160.528
C06943=1013.557,-117.499,-103.888,164.655,60.208,160.529
C06944=1013.552,-117.748,-103.880,164.652,60.214,160.529
C06945=1013.548,-118.029,-103.872,164.650,60.220,160.529
C06946=1013.542,-118.310,-103.864,164.646,60.226,160.529
C06947=1013.537,-118.591,-103.856,164.644,60.232,160.530
C06948=1013.531,-118.872,-103.849,164.641,60.237,160.530
C06949=1013.527,-119.121,-103.841,164.639,60.242,160.530
C06950=1013.523,-119.372,-103.835,164.636,60.248,160.530
C06951=1013.519,-119.621,-103.827,164.634,60.253,160.531
C06952=1013.514,-119.871,-103.821,164.631,60.258,160.531
C06953=1013.509,-120.122,-103.813,164.629,60.263,160.531
C06954=1013.504,-120.371,-103.806,164.627,60.268,160.531
C06955=1013.500,-120.621,-103.800,164.624,60.274,160.531
C06956=1013.495,-120.871,-103.792,164.621,60.279,160.532
C06957=1013.491,-121.121,-103.786,164.620,60.284,160.532
C06958=1013.486,-121.370,-103.779,164.616,60.288,160.532
C06959=1013.482,-121.621,-103.772,164.615,60.293,160.532
C06960=1013.478,-121.870,-103.765,164.612,60.299,160.532
C06961=1013.473,-122.120,-103.759,164.609,60.304,160.532
C06962=1013.469,-122.370,-103.751,164.607,60.309,160.533
C06963=1013.465,-122.620,-103.745,164.604,60.313,160.533
C06964=1013.459,-122.869,-103.738,164.602,60.318,160.533
C06965=1013.455,-123.120,-103.731,164.599,60.324,160.533
C06966=1013.451,-123.369,-103.724,164.598,60.328,160.533
C06967=1013.446,-123.619,-103.718,164.594,60.333,160.533
C06968=1013.442,-123.869,-103.710,164.592,60.338,160.533
C06969=1013.438,-124.119,-103.703,164.590,60.343,160.534
C06970=1013.433,-124.369,-103.697,164.587,60.349,160.534
C06971=1013.429,-124.619,-103.690,164.585,60.353,160.534
C06972=1013.425,-124.869,-103.683,164.582,60.358,160.534
C06973=1013.420,-125.118,-103.676,164.580,60.363,160.534
C06974=1013.416,-125.369,-103.670,164.577,60.368,160.534
C06975=1013.410,-125.618,-103.663,164.575,60.372,160.535
C06976=1013.406,-125.868,-103.656,164.572,60.378,160.535
C06977=1013.402,-126.118,-103.650,164.571,60.383,160.535
C06978=1013.397,-126.368,-103.643,164.567,60.387,160.535
C06979=1013.392,-126.618,-103.637,164.566,60.392,160.535
C06980=1013.388,-126.868,-103.630,164.562,60.397,160.535
C06981=1013.384,-127.118,-103.624,164.561,60.402,160.535
C06982=1013.379,-127.368,-103.617,164.559,60.406,160.536
C06983=1013.374,-127.617,-103.610,164.555,60.411,160.536
C06984=1013.370,-127.868,-103.604,164.554,60.416,160.536
C06985=1013.366,-128.116,-103.597,164.550,60.421,160.536
C06986=1013.362,-128.366,-103.590,164.549,60.425,160.536
C06987=1013.358,-128.616,-103.583,164.546,60.430,160.536
C06988=1013.354,-128.866,-103.575,164.544,60.434,160.536
C06989=1013.351,-129.115,-103.567,164.542,60.437,160.536
C06990=1013.347,-129.364,-103.558,164.538,60.439,160.535
C06991=1013.345,-129.614,-103.548,164.537,60.442,160.536
C06992=1013.342,-129.864,-103.537,164.535,60.444,160.535
C06993=1013.340,-130.114,-103.527,164.533,60.445,160.535
C06994=1013.339,-130.363,-103.514,164.529,60.446,160.534
C06995=1013.338,-130.613,-103.502,164.528,60.447,160.534
C06996=1013.336,-130.863,-103.490,164.526,60.448,160.533
C06997=1013.336,-131.112,-103.476,164.524,60.446,160.532
C06998=1013.336,-131.362,-103.462,164.522,60.446,160.532
C06999=1013.335,-131.612,-103.448,164.519,60.445,160.531
C07000=1013.336,-131.861,-103.433,164.518,60.444,160.530
C07001=1013.336,-132.111,-103.416,164.516,60.441,160.529
C07002=1013.338,-132.361,-103.401,164.514,60.439,160.528
C07003=1013.339,-132.610,-103.383,164.511,60.436,160.526
C07004=1013.341,-132.860,-103.366,164.509,60.433,160.525
C07005=1013.342,-133.110,-103.347,164.508,60.429,160.524
C07006=1013.345,-133.359,-103.328,164.505,60.425,160.522
C07007=1013.348,-133.609,-103.309,164.504,60.420,160.521
C07008=1013.351,-133.858,-103.289,164.501,60.415,160.519
C07009=1013.124,-133.884,-103.710,164.486,60.704,160.568
C07010=1013.121,-133.635,-103.730,164.489,60.708,160.570
C07011=1013.118,-133.386,-103.750,164.490,60.713,160.571
C07012=1013.116,-133.136,-103.768,164.492,60.717,160.573
C07013=1013.113,-132.886,-103.786,164.494,60.720,160.574
C07014=1013.112,-132.637,-103.804,164.496,60.724,160.575
C07015=1013.111,-132.387,-103.820,164.498,60.726,160.576
C07016=1013.110,-132.137,-103.838,164.500,60.728,160.577
C07017=1013.109,-131.887,-103.853,164.502,60.731,160.578
C07018=1013.108,-131.637,-103.868,164.505,60.732,160.579
C07019=1013.109,-131.388,-103.883,164.506,60.733,160.580
C07020=1013.109,-131.139,-103.897,164.508,60.734,160.581
C07021=1013.110,-130.889,-103.910,164.510,60.735,160.582
C07022=1013.111,-130.639,-103.924,164.512,60.734,160.582
C07023=1013.112,-130.389,-103.935,164.515,60.733,160.583
C07024=1013.113,-130.139,-103.947,164.518,60.733,160.584
C07025=1013.116,-129.890,-103.958,164.519,60.731,160.584
C07026=1013.118,-129.640,-103.968,164.521,60.730,160.585
C07027=1013.120,-129.391,-103.979,164.523,60.727,160.585
C07028=1013.123,-129.141,-103.987,164.526,60.725,160.585
C07029=1013.127,-128.892,-103.996,164.528,60.722,160.585
C07030=1013.130,-128.642,-104.004,164.531,60.718,160.585
C07031=1013.134,-128.393,-104.011,164.533,60.714,160.585
C07032=1013.139,-128.143,-104.018,164.535,60.710,160.585
C07033=1013.143,-127.893,-104.024,164.538,60.706,160.585
C07034=1013.147,-127.644,-104.031,164.539,60.701,160.585
C07035=1013.152,-127.394,-104.037,164.542,60.697,160.585
C07036=1013.156,-127.144,-104.044,164.545,60.692,160.585
C07037=1013.161,-126.894,-104.050,164.547,60.688,160.585
C07038=1013.165,-126.645,-104.058,164.549,60.683,160.585
C07039=1013.170,-126.395,-104.064,164.551,60.679,160.585
C07040=1013.174,-126.144,-104.070,164.554,60.675,160.585
C07041=1013.179,-125.894,-104.077,164.556,60.670,160.584
C07042=1013.183,-125.645,-104.084,164.559,60.666,160.584
C07043=1013.188,-125.395,-104.090,164.560,60.661,160.584
C07044=1013.192,-125.145,-104.097,164.564,60.656,160.584
C07045=1013.197,-124.895,-104.104,164.566,60.652,160.584
C07046=1013.201,-124.645,-104.110,164.568,60.647,160.584
C07047=1013.205,-124.395,-104.118,164.570,60.643,160.584
C07048=1013.210,-124.145,-104.124,164.574,60.638,160.584
C07049=1013.214,-123.895,-104.130,164.575,60.633,160.584
C07050=1013.219,-123.646,-104.138,164.577,60.629,160.584
C07051=1013.223,-123.396,-104.144,164.580,60.624,160.583
C07052=1013.228,-123.146,-104.151,164.583,60.620,160.583
C07053=1013.232,-122.896,-104.158,164.584,60.615,160.583
C07054=1013.237,-122.646,-104.165,164.588,60.610,160.583
C07055=1013.241,-122.396,-104.171,164.590,60.606,160.583
C07056=1013.245,-122.146,-104.178,164.592,60.601,160.583
C07057=1013.250,-121.897,-104.185,164.595,60.597,160.583
C07058=1013.254,-121.646,-104.192,164.597,60.592,160.583
C07059=1013.259,-121.397,-104.199,164.599,60.586,160.582
C07060=1013.263,-121.147,-104.205,164.602,60.582,160.582
C07061=1013.268,-120.897,-104.213,164.603,60.577,160.582
C07062=1013.272,-120.647,-104.220,164.607,60.573,160.582
C07063=1013.277,-120.398,-104.226,164.608,60.568,160.582
C07064=1013.281,-120.148,-104.233,164.612,60.563,160.582
C07065=1013.285,-119.898,-104.240,164.613,60.558,160.582
C07066=1013.290,-119.648,-104.248,164.616,60.553,160.581
C07067=1013.294,-119.398,-104.254,164.619,60.549,160.581
C07068=1013.299,-119.148,-104.261,164.621,60.543,160.581
C07069=1013.303,-118.898,-104.268,164.624,60.539,160.581
C07070=1013.308,-118.617,-104.275,164.626,60.533,160.581
C07071=1013.313,-118.336,-104.284,164.628,60.528,160.581
C07072=1013.318,-118.056,-104.291,164.631,60.522,160.580
C07073=1013.323,-117.775,-104.299,164.634,60.517,160.580
C07074=1013.328,-117.526,-104.306,164.637,60.512,160.580
C07075=1013.332,-117.276,-104.314,164.639,60.508,160.580
C07076=1013.337,-117.025,-104.320,164.642,60.502,160.580
C07077=1013.342,-116.776,-104.328,164.643,60.497,160.580
C07078=1013.346,-116.526,-104.335,164.646,60.492,160.579
C07079=1013.350,-116.276,-104.342,164.649,60.487,160.580
C07080=1013.355,-116.026,-104.349,164.651,60.483,160.579
C07081=1013.360,-115.777,-104.356,164.654,60.477,160.579
C07082=1013.364,-115.527,-104.363,164.656,60.472,160.579
C07083=1013.369,-115.276,-104.370,164.658,60.467,160.579
C07084=1013.374,-115.027,-104.377,164.662,60.462,160.579
C07085=1013.378,-114.777,-104.385,164.663,60.457,160.578
C07086=1013.382,-114.527,-104.391,164.666,60.452,160.578
C07087=1013.386,-114.277,-104.399,164.668,60.447,160.578
C07088=1013.391,-114.028,-104.406,164.670,60.442,160.578
C07089=1013.396,-113.777,-104.414,164.673,60.437,160.578
C07090=1013.400,-113.528,-104.421,164.676,60.432,160.578
C07091=1013.404,-113.278,-104.428,164.678,60.427,160.577
C07092=1013.409,-113.028,-104.435,164.681,60.422,160.577
C07093=1013.414,-112.779,-104.442,164.683,60.417,160.577
C07094=1013.419,-112.528,-104.450,164.685,60.411,160.577
C07095=1013.423,-112.279,-104.457,164.688,60.406,160.577
C07096=1013.427,-112.029,-104.465,164.690,60.401,160.576
C07097=1013.431,-111.779,-104.471,164.693,60.396,160.576
C07098=1013.436,-111.528,-104.479,164.695,60.391,160.576
C07099=1013.441,-111.279,-104.487,164.697,60.386,160.575
C07100=1013.446,-111.029,-104.493,164.700,60.380,160.575
C07101=1013.450,-110.780,-104.501,164.702,60.375,160.575
C07102=1013.455,-110.529,-104.509,164.705,60.370,160.575
C07103=1013.459,-110.280,-104.516,164.707,60.365,160.575
C07104=1013.464,-110.030,-104.523,164.710,60.359,160.574
C07105=1013.468,-109.780,-104.530,164.712,60.354,160.574
C07106=1013.473,-109.530,-104.538,164.715,60.349,160.574
C07107=1013.477,-109.280,-104.545,164.718,60.343,160.574
C07108=1013.482,-109.030,-104.553,164.720,60.339,160.574
C07109=1013.487,-108.781,-104.559,164.722,60.333,160.573
C07110=1013.492,-108.531,-104.567,164.725,60.328,160.573
C07111=1013.496,-108.281,-104.575,164.727,60.322,160.573
C07112=1013.500,-108.031,-104.582,164.730,60.316,160.573
C07113=1013.505,-107.781,-104.590,164.733,60.311,160.573
C07114=1013.510,-107.531,-104.597,164.734,60.306,160.572
C07115=1013.514,-107.282,-104.605,164.737,60.301,160.572
C07116=1013.519,-107.032,-104.612,164.740,60.296,160.572
C07117=1013.523,-106.782,-104.620,164.743,60.290,160.572
C07118=1013.528,-106.532,-104.627,164.745,60.284,160.571
C07119=1013.533,-106.282,-104.635,164.747,60.279,160.571
C07120=1013.537,-106.032,-104.642,164.749,60.274,160.571
C07121=1013.542,-105.783,-104.650,164.752,60.269,160.570
C07122=1013.546,-105.533,-104.659,164.755,60.263,160.570
C07123=1013.550,-105.283,-104.666,164.757,60.258,160.570
C07124=1013.555,-105.033,-104.674,164.759,60.252,160.570
C07125=1013.560,-104.783,-104.681,164.762,60.246,160.570
C07126=1013.564,-104.533,-104.689,164.765,60.241,160.569
C07127=1013.569,-104.283,-104.697,164.768,60.236,160.569
C07128=1013.573,-104.034,-104.705,164.770,60.230,160.569
C07129=1013.578,-103.784,-104.712,164.771,60.225,160.568
C07130=1013.583,-103.534,-104.720,164.774,60.220,160.568
C07131=1013.587,-103.284,-104.727,164.777,60.214,160.568
C07132=1013.592,-103.034,-104.735,164.779,60.208,160.568
C07133=1013.597,-102.785,-104.743,164.782,60.203,160.567
C07134=1013.602,-102.504,-104.751,164.785,60.196,160.567
C07135=1013.607,-102.224,-104.760,164.787,60.190,160.567
C07136=1013.612,-101.943,-104.769,164.790,60.184,160.566
C07137=1013.617,-101.663,-104.778,164.793,60.177,160.566
C07138=1013.622,-101.413,-104.785,164.796,60.172,160.566
C07139=1013.627,-101.163,-104.793,164.798,60.166,160.565
C07140=1013.631,-100.914,-104.801,164.801,60.160,160.565
C07141=1013.636,-100.663,-104.810,164.804,60.155,160.565
C07142=1013.640,-100.413,-104.817,164.806,60.149,160.565
C07143=1013.645,-100.163,-104.825,164.809,60.144,160.564
C07144=1013.649,-99.914,-104.833,164.811,60.138,160.564
C07145=1013.654,-99.664,-104.841,164.813,60.132,160.564
